KUKA KRL program: MyProgram_052().src

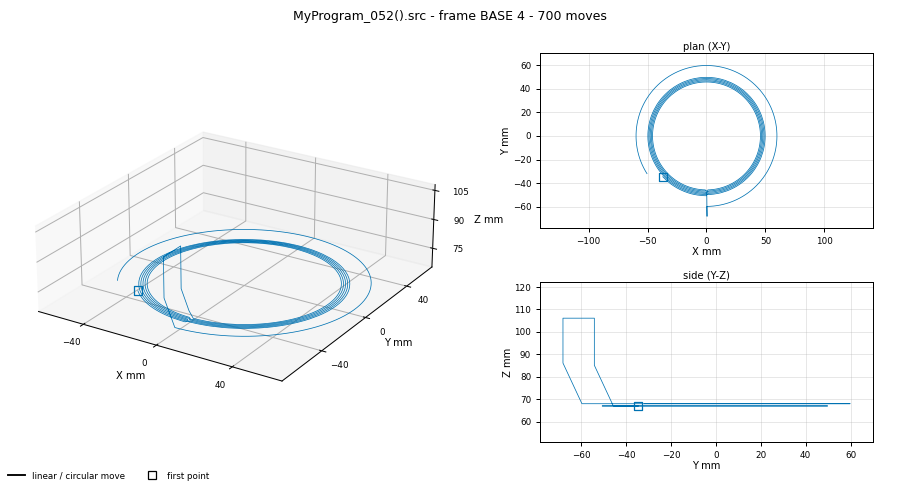
[picture p0: tool path of MyProgram_052().src in frame BASE 4, 700 of 700 moves have a stored position in this frame; points joined in program order, loops and branches not executed]
&ACCESS RVP
&REL 1
&PARAM TEMPLATE = C:\KRC\Roboter\Template\vorgabe
&PARAM EDITMASK = *
DEF MyProgram_052()
; ---- Setting reference (Base) ----
$BASE = BASE_DATA[4]

; --------------------------
; ---- Setting tool (TCP) ----
$TOOL = TOOL_DATA[3]
; --------------------------

$VEL.CP = VEL_APROX_PRINT
Startdeposition()
$VEL.CP = VEL_PRINT
LIN {X -37.0795,Y -34.6003,Z 67,A -142.3469,B 24.875,C -2.5805,E1 24.8845,E2 225.9733} C_DIS
LIN {X -35.1143,Y -36.5928,Z 67,A -139.506,B 24.8761,C -2.569,E1 24.8901,E2 223.1477} C_DIS
LIN {X -33.8275,Y -37.7853,Z 67,A -136.4507,B 24.8748,C -2.5821,E1 24.8966,E2 220.0491} C_DIS
LIN {X -30.4559,Y -40.5521,Z 67,A -131.9027,B 24.8763,C -2.5673,E1 24.9065,E2 215.5196} C_DIS
LIN {X -28.4082,Y -42.012,Z 67,A -128.4137,B 24.8757,C -2.5733,E1 24.9146,E2 212.0046} C_DIS
LIN {X -25.1167,Y -44.0592,Z 67,A -124.6294,B 24.8772,C -2.5574,E1 24.9237,E2 208.2469} C_DIS
LIN {X -22.6582,Y -45.3725,Z 67,A -121.2779,B 24.8772,C -2.5569,E1 24.9321,E2 204.8875} C_DIS
LIN {X -18.9408,Y -47.0459,Z 67,A -117.2171,B 24.8786,C -2.543,E1 24.9424,E2 200.8503} C_DIS
LIN {X -15.4527,Y -48.304,Z 67,A -112.4749,B 24.878,C -2.5491,E1 24.955,E2 196.0848} C_DIS
LIN {X -12.4723,Y -49.1576,Z 67,A -109.5038,B 24.8791,C -2.5379,E1 24.963,E2 193.1358} C_DIS
LIN {X -10.0949,Y -49.7005,Z 67,A -106.7826,B 24.8793,C -2.5361,E1 24.9704,E2 190.4157} C_DIS
LIN {X -7.4445,Y -50.1668,Z 67,A -103.2112,B 24.8785,C -2.5445,E1 24.9803,E2 186.8209} C_DIS
LIN {X -3.8911,Y -50.566,Z 67,A -100.05,B 24.88,C -2.5287,E1 24.989,E2 183.6956} C_DIS
LIN {X -2.1608,Y -50.6692,Z 67,A -97.7826,B 24.8794,C -2.5343,E1 24.9954,E2 181.4142} C_DIS
LIN {X -0.0557,Y -50.7153,Z 67,A -95.0288,B 24.8787,C -2.5416,E1 25.0031,E2 178.6432} C_DIS
LIN {X -0.0557,Y -50.7153,Z 67,A -95.0288,B 24.8787,C -2.5416,E1 25.0031,E2 178.6432} C_DIS
Enddeposition()
LIN {X 0.2505,Y -49.712,Z 67,A -95.9238,B 24.8792,C -2.5369,E1 25.0006,E2 179.5492} C_DIS
Startdeposition()
$VEL.CP = VEL_PRINT
LIN {X -2.7584,Y -49.6512,Z 67,A -99.9248,B 24.8801,C -2.5271,E1 24.9893,E2 183.5742} C_DIS
LIN {X -5.4391,Y -49.4301,Z 67,A -103.33,B 24.8806,C -2.5222,E1 24.9798,E2 186.9929} C_DIS
LIN {X -8.5864,Y -48.9804,Z 67,A -106.9223,B 24.8804,C -2.5244,E1 24.9699,E2 190.5832} C_DIS
LIN {X -12.0306,Y -48.2498,Z 67,A -110.567,B 24.8795,C -2.5331,E1 24.96,E2 194.212} C_DIS
LIN {X -15.2046,Y -47.3461,Z 67,A -115.2738,B 24.8807,C -2.5212,E1 24.9474,E2 198.9551} C_DIS
LIN {X -18.426,Y -46.1887,Z 67,A -119.1015,B 24.8802,C -2.5266,E1 24.9374,E2 202.778} C_DIS
LIN {X -22.1318,Y -44.5313,Z 67,A -122.9001,B 24.8783,C -2.5457,E1 24.9279,E2 206.5407} C_DIS
LIN {X -24.1155,Y -43.4892,Z 67,A -125.7875,B 24.8785,C -2.5443,E1 24.9208,E2 209.4396} C_DIS
LIN {X -27.878,Y -41.1784,Z 67,A -130.7372,B 24.8775,C -2.554,E1 24.9091,E2 214.382} C_DIS
LIN {X -29.9202,Y -39.7194,Z 67,A -133.864,B 24.8775,C -2.5552,E1 24.902,E2 217.5167} C_DIS
LIN {X -32.5332,Y -37.6097,Z 67,A -137.9216,B 24.877,C -2.5596,E1 24.8933,E2 221.5795} C_DIS
LIN {X -34.8779,Y -35.4455,Z 67,A -141.2483,B 24.8758,C -2.5721,E1 24.8866,E2 224.89} C_DIS
LIN {X -36.3763,Y -33.9066,Z 67,A -143.7227,B 24.8753,C -2.5774,E1 24.8819,E2 227.3625} C_DIS
LIN {X -37.7342,Y -32.3879,Z 67,A -145.936,B 24.8746,C -2.5845,E1 24.8778,E2 229.5687} C_DIS
LIN {X -38.7362,Y -31.183,Z 67,A -147.9222,B 24.8744,C -2.586,E1 24.8743,E2 231.5605} C_DIS
LIN {X -40.0423,Y -29.4865,Z 67,A -150.6165,B 24.8742,C -2.5886,E1 24.8697,E2 234.2615} C_DIS
LIN {X -42.0176,Y -26.5964,Z 67,A -154.4152,B 24.8729,C -2.6021,E1 24.8639,E2 238.0472} C_DIS
LIN {X -43.0644,Y -24.866,Z 67,A -157.367,B 24.8731,C -2.5994,E1 24.8597,E2 241.0208} C_DIS
LIN {X -44.6109,Y -21.9712,Z 67,A -160.8306,B 24.8717,C -2.614,E1 24.8553,E2 244.4679} C_DIS
LIN {X -45.6108,Y -19.8118,Z 67,A -163.4943,B 24.8708,C -2.6227,E1 24.8523,E2 247.1254} C_DIS
LIN {X -46.7007,Y -17.085,Z 67,A -166.8132,B 24.8698,C -2.6333,E1 24.849,E2 250.4376} C_DIS
LIN {X -47.5107,Y -14.6828,Z 67,A -170.2157,B 24.8696,C -2.6352,E1 24.8461,E2 253.855} C_DIS
LIN {X -48.4975,Y -10.9946,Z 67,A -173.9722,B 24.8674,C -2.6572,E1 24.8435,E2 257.5809} C_DIS
LIN {X -49.0589,Y -8.1285,Z 67,A -177.9765,B 24.8673,C -2.6587,E1 24.8415,E2 261.6052} C_DIS
LIN {X -49.4497,Y -5.2517,Z 67,A 179.0895,B 24.8657,C -2.6747,E1 24.8405,E2 264.5187} C_DIS
LIN {X -49.6264,Y -3.1776,Z 67,A 176.7448,B 24.8648,C -2.6829,E1 24.84,E2 266.8579} C_DIS
LIN {X -49.7186,Y -0.9552,Z 67,A 174.1077,B 24.8641,C -2.6899,E1 24.8398,E2 269.4941} C_DIS
LIN {X -49.6949,Y 1.8152,Z 67,A 170.5176,B 24.8636,C -2.6946,E1 24.84,E2 273.0947} C_DIS
LIN {X -49.522,Y 4.5195,Z 67,A 168.0202,B 24.8618,C -2.7128,E1 24.8405,E2 275.5633} C_DIS
LIN {X -49.2022,Y 7.208,Z 67,A 164.8184,B 24.8609,C -2.7215,E1 24.8416,E2 278.7635} C_DIS
LIN {X -48.9547,Y 8.7343,Z 67,A 162.6439,B 24.8609,C -2.7218,E1 24.8427,E2 280.9503} C_DIS
LIN {X -48.3657,Y 11.5613,Z 67,A 159.4302,B 24.8596,C -2.7336,E1 24.8446,E2 284.1545} C_DIS
LIN {X -47.5221,Y 14.646,Z 67,A 155.3988,B 24.859,C -2.7403,E1 24.8477,E2 288.1934} C_DIS
LIN {X -46.7485,Y 16.9539,Z 67,A 152.6347,B 24.858,C -2.7493,E1 24.8503,E2 290.9515} C_DIS
LIN {X -45.6266,Y 19.7752,Z 67,A 149.3564,B 24.8566,C -2.7627,E1 24.8538,E2 294.2159} C_DIS
LIN {X -44.6749,Y 21.8416,Z 67,A 146.0399,B 24.8568,C -2.7609,E1 24.8578,E2 297.5548} C_DIS
LIN {X -42.2626,Y 26.2058,Z 67,A 141.1281,B 24.8539,C -2.7886,E1 24.8646,E2 302.4259} C_DIS
LIN {X -40.6911,Y 28.5857,Z 67,A 136.9092,B 24.8544,C -2.7846,E1 24.8713,E2 306.6754} C_DIS
LIN {X -38.1447,Y 31.9031,Z 67,A 132.7078,B 24.8521,C -2.8056,E1 24.8785,E2 310.8463} C_DIS
LIN {X -36.5879,Y 33.6776,Z 67,A 130.0979,B 24.8513,C -2.8139,E1 24.8834,E2 313.448} C_DIS
LIN {X -35.0889,Y 35.2371,Z 67,A 127.5196,B 24.8508,C -2.8186,E1 24.8884,E2 316.0261} C_DIS
LIN {X -32.5963,Y 37.5546,Z 67,A 123.9843,B 24.8492,C -2.833,E1 24.8957,E2 319.5411} C_DIS
LIN {X -30.6979,Y 39.1218,Z 67,A 120.4276,B 24.8497,C -2.8286,E1 24.9035,E2 323.1218} C_DIS
LIN {X -28.804,Y 40.5362,Z 67,A 118.2528,B 24.8482,C -2.8421,E1 24.9083,E2 325.272} C_DIS
LIN {X -27.41,Y 41.4915,Z 67,A 115.4118,B 24.8493,C -2.8327,E1 24.915,E2 328.1448} C_DIS
LIN {X -23.7122,Y 43.7101,Z 67,A 110.8548,B 24.8477,C -2.8474,E1 24.926,E2 332.6803} C_DIS
LIN {X -20.8368,Y 45.1517,Z 67,A 107.4073,B 24.8466,C -2.857,E1 24.9346,E2 336.1138} C_DIS
LIN {X -18.9605,Y 45.9717,Z 67,A 104.6634,B 24.8469,C -2.8545,E1 24.9417,E2 338.87} C_DIS
LIN {X -15.5886,Y 47.2218,Z 67,A 100.8064,B 24.8459,C -2.864,E1 24.9518,E2 342.712} C_DIS
LIN {X -12.4514,Y 48.1437,Z 67,A 96.9923,B 24.8456,C -2.8672,E1 24.962,E2 346.5245} C_DIS
LIN {X -10.0971,Y 48.6919,Z 67,A 94.2114,B 24.8453,C -2.8696,E1 24.9696,E2 349.303} C_DIS
LIN {X -7.651,Y 49.1354,Z 67,A 91.5672,B 24.8447,C -2.8752,E1 24.9769,E2 351.9365} C_DIS
LIN {X -5.9044,Y 49.3761,Z 67,A 89.1599,B 24.8452,C -2.8703,E1 24.9836,E2 354.357} C_DIS
LIN {X -2.8923,Y 49.6437,Z 67,A 85.7598,B 24.8449,C -2.8732,E1 24.993,E2 357.7518} C_DIS
LIN {X -0.6646,Y 49.7234,Z 67,A 82.8665,B 24.8454,C -2.8686,E1 25.0011,E2 360.6563} C_DIS
LIN {X 2.8209,Y 49.6477,Z 67,A 78.8494,B 24.8454,C -2.8688,E1 25.0123,E2 364.6716} C_DIS
LIN {X 6.9409,Y 49.241,Z 67,A 75.0745,B 24.8436,C -2.8849,E1 25.0227,E2 368.4058} C_DIS
LIN {X 8.9379,Y 48.9175,Z 67,A 72.2375,B 24.8446,C -2.8755,E1 25.0306,E2 371.2623} C_DIS
LIN {X 12.2001,Y 48.2076,Z 67,A 67.5135,B 24.8465,C -2.8584,E1 25.0435,E2 376.0201} C_DIS
LIN {X 15.4724,Y 47.2597,Z 67,A 63.7622,B 24.8465,C -2.8584,E1 25.0535,E2 379.7645} C_DIS
LIN {X 19.2501,Y 45.8507,Z 67,A 60.0313,B 24.8452,C -2.8701,E1 25.0631,E2 383.4594} C_DIS
LIN {X 20.5782,Y 45.2704,Z 67,A 58.1872,B 24.8458,C -2.8651,E1 25.0678,E2 385.3108} C_DIS
LIN {X 22.4752,Y 44.3592,Z 67,A 54.4297,B 24.8486,C -2.8384,E1 25.0773,E2 389.1215} C_DIS
LIN {X 25.4752,Y 42.7072,Z 67,A 52.1521,B 24.846,C -2.8629,E1 25.0826,E2 391.3341} C_DIS
LIN {X 28.0765,Y 41.0441,Z 67,A 48.3054,B 24.8472,C -2.8521,E1 25.0917,E2 395.1939} C_DIS
LIN {X 29.9486,Y 39.6981,Z 67,A 45.4003,B 24.8482,C -2.843,E1 25.0982,E2 398.1102} C_DIS
LIN {X 32.0395,Y 38.0315,Z 67,A 41.483,B 24.8504,C -2.8218,E1 25.1067,E2 402.0627} C_DIS
LIN {X 34.3865,Y 35.9228,Z 67,A 37.8471,B 24.8512,C -2.8144,E1 25.1141,E2 405.701} C_DIS
LIN {X 37.3665,Y 32.8115,Z 67,A 33.7329,B 24.8507,C -2.8195,E1 25.1218,E2 409.7849} C_DIS
LIN {X 39.222,Y 30.5701,Z 67,A 30.767,B 24.8507,C -2.8192,E1 25.1269,E2 412.738} C_DIS
LIN {X 40.1847,Y 29.2925,Z 67,A 28.2929,B 24.8525,C -2.8026,E1 25.1311,E2 415.2393} C_DIS
LIN {X 42.0752,Y 26.5059,Z 67,A 24.9676,B 24.8524,C -2.8035,E1 25.1361,E2 418.5458} C_DIS
LIN {X 43.2785,Y 24.4929,Z 67,A 21.1417,B 24.8554,C -2.7747,E1 25.1415,E2 422.4201} C_DIS
LIN {X 44.8673,Y 21.4426,Z 67,A 17.9731,B 24.8549,C -2.7793,E1 25.1454,E2 425.5609} C_DIS
LIN {X 46.0689,Y 18.7215,Z 67,A 14.8326,B 24.8553,C -2.7753,E1 25.1488,E2 428.6938} C_DIS
LIN {X 46.7802,Y 16.8668,Z 67,A 12.2733,B 24.8566,C -2.7633,E1 25.1513,E2 431.267} C_DIS
LIN {X 47.7862,Y 13.7604,Z 67,A 9.0045,B 24.8567,C -2.762,E1 25.1539,E2 434.5203} C_DIS
LIN {X 48.2557,Y 12.0119,Z 67,A 6.634,B 24.8579,C -2.7501,E1 25.1556,E2 436.9052} C_DIS
LIN {X 48.8256,Y 9.4293,Z 67,A 3.4803,B 24.8591,C -2.7387,E1 25.1574,E2 440.0675} C_DIS
LIN {X 49.299,Y 6.5169,Z 67,A 0.1433,B 24.8601,C -2.7295,E1 25.1587,E2 443.4067} C_DIS
LIN {X 49.599,Y 3.5824,Z 67,A -3.0614,B 24.8608,C -2.7228,E1 25.1595,E2 446.6083} C_DIS
LIN {X 49.7259,Y 0.5187,Z 67,A -6.1684,B 24.861,C -2.7203,E1 25.1598,E2 449.7027} C_DIS
LIN {X 49.6721,Y -2.3404,Z 67,A -10.1157,B 24.8634,C -2.6968,E1 25.1594,E2 453.6821} C_DIS
LIN {X 49.4176,Y -5.5441,Z 67,A -13.6854,B 24.8643,C -2.6878,E1 25.1585,E2 457.2519} C_DIS
LIN {X 49.0237,Y -8.3395,Z 67,A -16.716,B 24.8649,C -2.682,E1 25.1572,E2 460.2784} C_DIS
LIN {X 48.5542,Y -10.7407,Z 67,A -19.5373,B 24.8658,C -2.6731,E1 25.1556,E2 463.1042} C_DIS
LIN {X 47.9955,Y -13.0107,Z 67,A -22.9399,B 24.8681,C -2.6507,E1 25.1531,E2 466.5404} C_DIS
LIN {X 46.3058,Y -18.128,Z 67,A -28.0338,B 24.8677,C -2.654,E1 25.1485,E2 471.5977} C_DIS
LIN {X 45.2339,Y -20.6589,Z 67,A -32.1672,B 24.8706,C -2.6254,E1 25.1438,E2 475.7762} C_DIS
LIN {X 43.2933,Y -24.4656,Z 67,A -36.6993,B 24.8712,C -2.619,E1 25.1378,E2 480.2998} C_DIS
LIN {X 41.4212,Y -27.5166,Z 67,A -40.1738,B 24.8711,C -2.6203,E1 25.1327,E2 483.7534} C_DIS
LIN {X 40.6509,Y -28.6409,Z 67,A -42.2645,B 24.8725,C -2.6059,E1 25.1293,E2 485.8682} C_DIS
LIN {X 38.573,Y -31.3844,Z 67,A -45.7048,B 24.8725,C -2.6057,E1 25.1234,E2 489.2925} C_DIS
LIN {X 36.6935,Y -33.5625,Z 67,A -49.7313,B 24.8747,C -2.5836,E1 25.1159,E2 493.3535} C_DIS
LIN {X 34.5074,Y -35.8063,Z 67,A -53.3041,B 24.8754,C -2.5757,E1 25.1088,E2 496.9298} C_DIS
LIN {X 31.3977,Y -38.5622,Z 67,A -57.3951,B 24.8752,C -2.5784,E1 25.1002,E2 500.9984} C_DIS
LIN {X 29.3776,Y -40.1224,Z 67,A -60.7741,B 24.8766,C -2.564,E1 25.0926,E2 504.3994} C_DIS
LIN {X 27.4879,Y -41.4401,Z 67,A -62.9553,B 24.8762,C -2.5677,E1 25.0876,E2 506.5643} C_DIS
LIN {X 25.4166,Y -42.7418,Z 67,A -66.3813,B 24.8778,C -2.5512,E1 25.0794,E2 510.0189} C_DIS
LIN {X 23.1942,Y -43.9872,Z 67,A -68.7496,B 24.8773,C -2.5567,E1 25.0736,E2 512.3672} C_DIS
LIN {X 19.9272,Y -45.5605,Z 67,A -73.7738,B 24.8794,C -2.5348,E1 25.0608,E2 517.4306} C_DIS
LIN {X 17.454,Y -46.5643,Z 67,A -77.1022,B 24.8802,C -2.5261,E1 25.0521,E2 520.7725} C_DIS
LIN {X 12.1079,Y -48.2312,Z 67,A -82.4712,B 24.879,C -2.5385,E1 25.0378,E2 526.1029} C_DIS
LIN {X 10.0818,Y -48.6949,Z 67,A -85.0863,B 24.8796,C -2.5324,E1 25.0306,E2 528.729} C_DIS
LIN {X 7.4223,Y -49.171,Z 67,A -87.7994,B 24.8792,C -2.5372,E1 25.0232,E2 531.428} C_DIS
LIN {X 6.033,Y -49.3603,Z 67,A -89.9034,B 24.8801,C -2.5276,E1 25.0173,E2 533.5531} C_DIS
LIN {X 3.1793,Y -49.6263,Z 67,A -93.4479,B 24.8806,C -2.5219,E1 25.0074,E2 537.1095} C_DIS
LIN {X 0.2505,Y -49.712,Z 67,A -95.9232,B 24.8792,C -2.5367,E1 25.0006,E2 539.5492} C_DIS
Enddeposition()
LIN {X 0.2505,Y -49.712,Z 67,A -95.9232,B 24.8792,C -2.5367,E1 25.0006,E2 539.5492} C_DIS
Startdeposition()
$VEL.CP = VEL_PRINT
LIN {X 1.4593,Y -48.7184,Z 67,A -93.5201,B 24.8759,C -2.5709,E1 25.0075,E2 537.0653} C_DIS
LIN {X 3.9754,Y -48.5779,Z 67,A -90.7627,B 24.8761,C -2.5686,E1 25.0152,E2 534.3145} C_DIS
LIN {X 6.1747,Y -48.3476,Z 67,A -88.2241,B 24.8761,C -2.5691,E1 25.0222,E2 531.7766} C_DIS
LIN {X 9.1506,Y -47.8736,Z 67,A -83.9458,B 24.8746,C -2.5849,E1 25.034,E2 527.4652} C_DIS
LIN {X 14.099,Y -46.6564,Z 67,A -77.8877,B 24.8738,C -2.5924,E1 25.0504,E2 521.3992} C_DIS
LIN {X 17.6898,Y -45.417,Z 67,A -73.6014,B 24.8736,C -2.5949,E1 25.0616,E2 517.116} C_DIS
LIN {X 21.6587,Y -43.6636,Z 67,A -69.008,B 24.8737,C -2.5933,E1 25.0732,E2 512.5382} C_DIS
LIN {X 24.0511,Y -42.3932,Z 67,A -65.7906,B 24.8731,C -2.5993,E1 25.0811,E2 509.3158} C_DIS
LIN {X 26.2006,Y -41.0994,Z 67,A -62.4617,B 24.8719,C -2.612,E1 25.089,E2 505.9674} C_DIS
LIN {X 29.7642,Y -38.5967,Z 67,A -57.7772,B 24.8717,C -2.6141,E1 25.0995,E2 501.2945} C_DIS
LIN {X 32.7938,Y -36.0568,Z 67,A -52.8175,B 24.8701,C -2.6305,E1 25.11,E2 496.3155} C_DIS
LIN {X 35.5576,Y -33.3335,Z 67,A -47.8569,B 24.8682,C -2.6494,E1 25.1197,E2 491.3315} C_DIS
LIN {X 38.127,Y -30.364,Z 67,A -43.4377,B 24.8674,C -2.6573,E1 25.1275,E2 486.9139} C_DIS
LIN {X 40.6831,Y -26.842,Z 67,A -38.9979,B 24.8674,C -2.6578,E1 25.1346,E2 482.4949} C_DIS
LIN {X 42.0184,Y -24.6997,Z 67,A -36.0839,B 24.8666,C -2.665,E1 25.1388,E2 479.5785} C_DIS
LIN {X 43.3733,Y -22.2345,Z 67,A -33.2124,B 24.8666,C -2.6659,E1 25.1426,E2 476.72} C_DIS
LIN {X 44.4214,Y -20.0587,Z 67,A -29.4695,B 24.8639,C -2.6923,E1 25.1471,E2 472.9349} C_DIS
LIN {X 45.6985,Y -16.9491,Z 67,A -25.6028,B 24.8628,C -2.7025,E1 25.151,E2 469.0656} C_DIS
LIN {X 46.9143,Y -13.216,Z 67,A -21.4414,B 24.8623,C -2.7075,E1 25.1544,E2 464.916} C_DIS
LIN {X 47.7125,Y -9.9576,Z 67,A -17.156,B 24.8604,C -2.7267,E1 25.157,E2 460.6102} C_DIS
LIN {X 48.2077,Y -7.1897,Z 67,A -14.3099,B 24.8603,C -2.7278,E1 25.1583,E2 457.7781} C_DIS
LIN {X 48.4802,Y -5.0283,Z 67,A -11.7765,B 24.8595,C -2.7353,E1 25.1591,E2 455.2419} C_DIS
LIN {X 48.6854,Y -2.3119,Z 67,A -8.1781,B 24.8576,C -2.7534,E1 25.1597,E2 451.6221} C_DIS
LIN {X 48.7412,Y 0.2134,Z 67,A -5.2697,B 24.8568,C -2.7615,E1 25.1597,E2 448.712} C_DIS
LIN {X 48.6356,Y 3.1938,Z 67,A -1.9945,B 24.8561,C -2.7678,E1 25.1593,E2 445.4412} C_DIS
LIN {X 48.4596,Y 5.2249,Z 67,A 0.2962,B 24.8555,C -2.7732,E1 25.1586,E2 443.1514} C_DIS
LIN {X 47.9146,Y 8.9375,Z 67,A 4.6496,B 24.8543,C -2.7855,E1 25.1567,E2 438.7943} C_DIS
LIN {X 47.2883,Y 11.8111,Z 67,A 8.1227,B 24.8531,C -2.7963,E1 25.1545,E2 435.3159} C_DIS
LIN {X 46.5524,Y 14.4391,Z 67,A 11.526,B 24.8517,C -2.8097,E1 25.1518,E2 431.9005} C_DIS
LIN {X 45.5852,Y 17.251,Z 67,A 14.5058,B 24.8517,C -2.8095,E1 25.149,E2 428.9376} C_DIS
LIN {X 44.771,Y 19.267,Z 67,A 17.3201,B 24.8504,C -2.8218,E1 25.146,E2 426.1097} C_DIS
LIN {X 43.9622,Y 21.0462,Z 67,A 19.3244,B 24.8504,C -2.8224,E1 25.1436,E2 424.1148} C_DIS
LIN {X 42.5457,Y 23.7797,Z 67,A 23.1875,B 24.8488,C -2.8369,E1 25.1386,E2 420.2378} C_DIS
LIN {X 41.3344,Y 25.8279,Z 67,A 25.7483,B 24.8485,C -2.8395,E1 25.1349,E2 417.6839} C_DIS
LIN {X 40.3728,Y 27.3066,Z 67,A 28.4737,B 24.8466,C -2.8573,E1 25.1306,E2 414.9297} C_DIS
LIN {X 38.5139,Y 29.8716,Z 67,A 32.2504,B 24.8455,C -2.8672,E1 25.1242,E2 411.1476} C_DIS
LIN {X 36.3063,Y 32.5187,Z 67,A 35.8708,B 24.8455,C -2.868,E1 25.1176,E2 407.5417} C_DIS
LIN {X 33.6815,Y 35.2308,Z 67,A 40.9102,B 24.8432,C -2.8887,E1 25.1076,E2 402.4747} C_DIS
LIN {X 30.8052,Y 37.7713,Z 67,A 44.786,B 24.8436,C -2.8852,E1 25.0994,E2 398.6222} C_DIS
LIN {X 28.1121,Y 39.8168,Z 67,A 48.2961,B 24.8438,C -2.8834,E1 25.0915,E2 395.1288} C_DIS
LIN {X 25.7687,Y 41.3714,Z 67,A 51.6887,B 24.8431,C -2.8901,E1 25.0836,E2 391.7315} C_DIS
LIN {X 24.4467,Y 42.1658,Z 67,A 53.8882,B 24.842,C -2.8997,E1 25.0782,E2 389.5159} C_DIS
LIN {X 21.4963,Y 43.7441,Z 67,A 57.6781,B 24.8417,C -2.9021,E1 25.0689,E2 385.7308} C_DIS
LIN {X 19.4392,Y 44.696,Z 67,A 60.07,B 24.842,C -2.9002,E1 25.0628,E2 383.3494} C_DIS
LIN {X 17.4937,Y 45.4922,Z 67,A 63.0781,B 24.8406,C -2.9121,E1 25.0549,E2 380.3197} C_DIS
LIN {X 14.4878,Y 46.5373,Z 67,A 66.272,B 24.8414,C -2.9055,E1 25.0465,E2 377.1476} C_DIS
LIN {X 12.305,Y 47.161,Z 67,A 69.2063,B 24.8407,C -2.9118,E1 25.0386,E2 374.203} C_DIS
LIN {X 9.7775,Y 47.7495,Z 67,A 72.2311,B 24.8406,C -2.9129,E1 25.0303,E2 371.1797} C_DIS
LIN {X 7.2536,Y 48.1976,Z 67,A 75.2551,B 24.8404,C -2.914,E1 25.022,E2 368.1561} C_DIS
LIN {X 4.5447,Y 48.5279,Z 67,A 78.6127,B 24.8401,C -2.917,E1 25.0127,E2 364.7937} C_DIS
LIN {X 1.7948,Y 48.7077,Z 67,A 81.8002,B 24.8402,C -2.916,E1 25.0038,E2 361.6096} C_DIS
LIN {X -0.4565,Y 48.7383,Z 67,A 84.1756,B 24.8408,C -2.911,E1 24.9972,E2 359.2462} C_DIS
LIN {X -2.6649,Y 48.6673,Z 67,A 86.9936,B 24.8405,C -2.9138,E1 24.9893,E2 356.4211} C_DIS
LIN {X -4.7797,Y 48.5057,Z 67,A 89.5773,B 24.8405,C -2.914,E1 24.9821,E2 353.8354} C_DIS
LIN {X -6.6855,Y 48.2795,Z 67,A 91.8359,B 24.8405,C -2.9127,E1 24.9759,E2 351.5782} C_DIS
LIN {X -9.959,Y 47.7122,Z 67,A 96.0485,B 24.8404,C -2.9145,E1 24.9643,E2 347.3566} C_DIS
LIN {X -14.1936,Y 46.6285,Z 67,A 100.7637,B 24.8417,C -2.9026,E1 24.9517,E2 342.6626} C_DIS
LIN {X -16.3104,Y 45.9305,Z 67,A 103.2846,B 24.8422,C -2.898,E1 24.945,E2 340.1479} C_DIS
LIN {X -18.2361,Y 45.2004,Z 67,A 106.0304,B 24.842,C -2.8997,E1 24.9379,E2 337.392} C_DIS
LIN {X -21.0515,Y 43.9595,Z 67,A 109.3865,B 24.843,C -2.8904,E1 24.9294,E2 334.0498} C_DIS
LIN {X -23.0132,Y 42.9659,Z 67,A 112.6518,B 24.8424,C -2.8964,E1 24.9213,E2 330.7611} C_DIS
LIN {X -27.1404,Y 40.4849,Z 67,A 117.4332,B 24.8449,C -2.873,E1 24.91,E2 326.0207} C_DIS
LIN {X -29.6729,Y 38.667,Z 67,A 122.0754,B 24.8442,C -2.8799,E1 24.8995,E2 321.3454} C_DIS
LIN {X -32.0865,Y 36.6888,Z 67,A 125.4244,B 24.8455,C -2.8672,E1 24.8925,E2 318.0138} C_DIS
LIN {X -34.5849,Y 34.3437,Z 67,A 128.9159,B 24.8474,C -2.8501,E1 24.8855,E2 314.5485} C_DIS
LIN {X -35.6779,Y 33.206,Z 67,A 131.5205,B 24.8467,C -2.8563,E1 24.8805,E2 311.9176} C_DIS
LIN {X -38.542,Y 29.8352,Z 67,A 135.6777,B 24.8497,C -2.8284,E1 24.8732,E2 307.8081} C_DIS
LIN {X -39.8556,Y 28.0576,Z 67,A 139.4151,B 24.8488,C -2.8374,E1 24.867,E2 304.031} C_DIS
LIN {X -41.2946,Y 25.8916,Z 67,A 141.8914,B 24.8505,C -2.8208,E1 24.8633,E2 301.5817} C_DIS
LIN {X -42.2826,Y 24.2435,Z 67,A 144.4806,B 24.8507,C -2.8191,E1 24.8597,E2 298.9832} C_DIS
LIN {X -43.9141,Y 21.1462,Z 67,A 148.3951,B 24.8523,C -2.8044,E1 24.8548,E2 295.0829} C_DIS
LIN {X -44.9155,Y 18.9264,Z 67,A 151.2125,B 24.8532,C -2.7953,E1 24.8516,E2 292.2717} C_DIS
LIN {X -45.8241,Y 16.6065,Z 67,A 153.896,B 24.8545,C -2.7831,E1 24.849,E2 289.6021} C_DIS
LIN {X -46.5695,Y 14.3838,Z 67,A 157.4063,B 24.8543,C -2.785,E1 24.846,E2 286.0673} C_DIS
LIN {X -47.4055,Y 11.3304,Z 67,A 160.3577,B 24.8566,C -2.763,E1 24.844,E2 283.1512} C_DIS
LIN {X -47.7895,Y 9.5786,Z 67,A 162.6746,B 24.857,C -2.7593,E1 24.8426,E2 280.8297} C_DIS
LIN {X -48.2667,Y 6.7781,Z 67,A 166.8386,B 24.857,C -2.7601,E1 24.8408,E2 276.639} C_DIS
LIN {X -48.6347,Y 3.2063,Z 67,A 170.7388,B 24.8587,C -2.7424,E1 24.84,E2 272.7577} C_DIS
LIN {X -48.7424,Y 0.0227,Z 67,A 174.5122,B 24.8599,C -2.731,E1 24.8398,E2 268.9889} C_DIS
LIN {X -48.6213,Y -3.4029,Z 67,A 178.1219,B 24.8618,C -2.7127,E1 24.8403,E2 265.4012} C_DIS
LIN {X -48.4408,Y -5.3948,Z 67,A -179.255,B 24.8622,C -2.7091,E1 24.841,E2 262.7709} C_DIS
LIN {X -48.0762,Y -8.0162,Z 67,A -176.3395,B 24.8634,C -2.6969,E1 24.8423,E2 259.8673} C_DIS
LIN {X -47.5785,Y -10.5799,Z 67,A -172.8888,B 24.8638,C -2.6928,E1 24.8442,E2 256.406} C_DIS
LIN {X -46.7055,Y -13.9359,Z 67,A -169.0415,B 24.8654,C -2.6775,E1 24.8471,E2 252.5729} C_DIS
LIN {X -45.9885,Y -16.1451,Z 67,A -166.1966,B 24.866,C -2.6711,E1 24.8496,E2 249.727} C_DIS
LIN {X -44.665,Y -19.5103,Z 67,A -161.662,B 24.8668,C -2.6631,E1 24.8545,E2 245.1864} C_DIS
LIN {X -43.2186,Y -22.5344,Z 67,A -157.8085,B 24.868,C -2.6512,E1 24.8593,E2 241.3407} C_DIS
LIN {X -41.6168,Y -25.3705,Z 67,A -153.8406,B 24.8688,C -2.6432,E1 24.8649,E2 237.3712} C_DIS
LIN {X -40.1943,Y -27.5702,Z 67,A -151.3138,B 24.8704,C -2.6276,E1 24.8688,E2 234.8692} C_DIS
LIN {X -38.8864,Y -29.3846,Z 67,A -148.356,B 24.8705,C -2.626,E1 24.8737,E2 231.9008} C_DIS
LIN {X -37.3702,Y -31.2907,Z 67,A -145.5748,B 24.8713,C -2.6183,E1 24.8786,E2 229.1253} C_DIS
LIN {X -35.6731,Y -33.2129,Z 67,A -142.3396,B 24.8716,C -2.615,E1 24.8847,E2 225.8837} C_DIS
LIN {X -33.8634,Y -35.0555,Z 67,A -139.6153,B 24.8727,C -2.6041,E1 24.89,E2 223.1737} C_DIS
LIN {X -32.2252,Y -36.5675,Z 67,A -136.7648,B 24.8728,C -2.6025,E1 24.896,E2 220.3158} C_DIS
LIN {X -30.3831,Y -38.112,Z 67,A -133.7171,B 24.873,C -2.6007,E1 24.9026,E2 217.2608} C_DIS
LIN {X -27.5312,Y -40.2207,Z 67,A -129.8182,B 24.8741,C -2.5897,E1 24.9114,E2 213.3746} C_DIS
LIN {X -24.555,Y -42.1039,Z 67,A -125.5983,B 24.8746,C -2.5849,E1 24.9215,E2 209.153} C_DIS
LIN {X -23.107,Y -42.915,Z 67,A -123.4273,B 24.8745,C -2.5858,E1 24.9268,E2 206.9737} C_DIS
LIN {X -20.4141,Y -44.2595,Z 67,A -119.7902,B 24.8747,C -2.5833,E1 24.936,E2 203.3333} C_DIS
LIN {X -17.4239,Y -45.5198,Z 67,A -116.5653,B 24.876,C -2.5702,E1 24.9443,E2 200.1325} C_DIS
LIN {X -15.5468,Y -46.1942,Z 67,A -113.8882,B 24.8757,C -2.5736,E1 24.9514,E2 197.442} C_DIS
LIN {X -12.8352,Y -47.02,Z 67,A -110.5462,B 24.8758,C -2.5716,E1 24.9604,E2 194.0994} C_DIS
LIN {X -9.4545,Y -47.8151,Z 67,A -105.9303,B 24.8752,C -2.5787,E1 24.973,E2 189.4611} C_DIS
LIN {X -5.6403,Y -48.4128,Z 67,A -101.9402,B 24.8761,C -2.5685,E1 24.984,E2 185.492} C_DIS
LIN {X -2.9306,Y -48.6526,Z 67,A -99.0645,B 24.8767,C -2.563,E1 24.992,E2 182.6282} C_DIS
LIN {X -1.0392,Y -48.7294,Z 67,A -96.7997,B 24.8766,C -2.564,E1 24.9983,E2 180.3608} C_DIS
LIN {X 0.2379,Y -48.7342,Z 67,A -95.3358,B 24.8766,C -2.5638,E1 25.0024,E2 178.8975} C_DIS
Enddeposition()
LIN {X 0.2379,Y -48.7342,Z 67,A -95.3358,B 24.8766,C -2.5638,E1 25.0024,E2 178.8975} C_DIS
Startdeposition()
$VEL.CP = VEL_PRINT
LIN {X -0.8805,Y -47.7446,Z 67,A -97.8451,B 24.8769,C -2.561,E1 24.9954,E2 181.4134} C_DIS
LIN {X -3.3224,Y -47.6371,Z 67,A -100.7978,B 24.8769,C -2.5605,E1 24.9871,E2 184.3681} C_DIS
LIN {X -5.768,Y -47.4036,Z 67,A -103.7394,B 24.8769,C -2.5609,E1 24.9789,E2 187.3105} C_DIS
LIN {X -8.6463,Y -46.9639,Z 67,A -107.7465,B 24.8776,C -2.5539,E1 24.9679,E2 191.3382} C_DIS
LIN {X -12.3361,Y -46.132,Z 67,A -111.6373,B 24.8764,C -2.5664,E1 24.9574,E2 195.2047} C_DIS
LIN {X -15.4067,Y -45.1994,Z 67,A -115.1387,B 24.8756,C -2.5745,E1 24.9481,E2 198.6927} C_DIS
LIN {X -17.9717,Y -44.2419,Z 67,A -118.9673,B 24.8761,C -2.5692,E1 24.938,E2 202.542} C_DIS
LIN {X -21.0789,Y -42.8489,Z 67,A -122.9705,B 24.8755,C -2.575,E1 24.9279,E2 206.5414} C_DIS
LIN {X -22.4857,Y -42.1282,Z 67,A -124.9714,B 24.8755,C -2.5759,E1 24.923,E2 208.5459} C_DIS
LIN {X -25.2515,Y -40.5301,Z 67,A -128.6188,B 24.8746,C -2.584,E1 24.9142,E2 212.1849} C_DIS
LIN {X -26.8598,Y -39.4827,Z 67,A -131.226,B 24.8747,C -2.5832,E1 24.9081,E2 214.8028} C_DIS
LIN {X -29.3649,Y -37.6577,Z 67,A -134.5088,B 24.8735,C -2.5958,E1 24.9008,E2 218.0671} C_DIS
LIN {X -31.275,Y -36.0862,Z 67,A -137.9785,B 24.8737,C -2.5941,E1 24.8934,E2 221.5541} C_DIS
LIN {X -33.3426,Y -34.1846,Z 67,A -141.3462,B 24.873,C -2.6009,E1 24.8866,E2 224.9196} C_DIS
LIN {X -34.97,Y -32.5192,Z 67,A -143.7846,B 24.8719,C -2.6118,E1 24.8819,E2 227.3426} C_DIS
LIN {X -36.4873,Y -30.8059,Z 67,A -146.7887,B 24.8717,C -2.6143,E1 24.8764,E2 230.3541} C_DIS
LIN {X -37.9974,Y -28.9223,Z 67,A -149.7426,B 24.8711,C -2.6203,E1 24.8713,E2 233.3077} C_DIS
LIN {X -39.0395,Y -27.5013,Z 67,A -151.7547,B 24.8704,C -2.6268,E1 24.8681,E2 235.3141} C_DIS
LIN {X -40.9376,Y -24.5855,Z 67,A -156.3462,B 24.8699,C -2.6319,E1 24.8612,E2 239.9169} C_DIS
LIN {X -42.3573,Y -22.0507,Z 67,A -159.1053,B 24.8681,C -2.6508,E1 24.8576,E2 242.6452} C_DIS
LIN {X -43.1053,Y -20.5493,Z 67,A -161.6755,B 24.8682,C -2.6489,E1 24.8544,E2 245.234} C_DIS
LIN {X -44.2989,Y -17.8315,Z 67,A -164.6864,B 24.8665,C -2.6662,E1 24.8511,E2 248.2202} C_DIS
LIN {X -45.2199,Y -15.3458,Z 67,A -168.2612,B 24.8661,C -2.6701,E1 24.8477,E2 251.8058} C_DIS
LIN {X -45.9403,Y -13.0314,Z 67,A -171.8862,B 24.8661,C -2.6695,E1 24.8449,E2 255.4534} C_DIS
LIN {X -46.6754,Y -10.0866,Z 67,A -175.843,B 24.8655,C -2.6764,E1 24.8425,E2 259.4167} C_DIS
LIN {X -47.5276,Y -4.6383,Z 67,A 177.5165,B 24.8634,C -2.6966,E1 24.8402,E2 266.0488} C_DIS
LIN {X -47.7544,Y 0.123,Z 67,A 172.5012,B 24.8607,C -2.7234,E1 24.8398,E2 271.03} C_DIS
LIN {X -47.6492,Y 3.1444,Z 67,A 168.9744,B 24.8594,C -2.7362,E1 24.8403,E2 274.5476} C_DIS
LIN {X -47.4199,Y 5.6286,Z 67,A 165.7581,B 24.8587,C -2.7427,E1 24.8412,E2 277.7674} C_DIS
LIN {X -46.9854,Y 8.5266,Z 67,A 162.3283,B 24.8575,C -2.7548,E1 24.8428,E2 281.1887} C_DIS
LIN {X -46.4595,Y 11.0418,Z 67,A 159.1989,B 24.8565,C -2.7638,E1 24.8447,E2 284.315} C_DIS
LIN {X -45.4398,Y 14.6815,Z 67,A 154.9667,B 24.8547,C -2.7816,E1 24.848,E2 288.5289} C_DIS
LIN {X -44.837,Y 16.4309,Z 67,A 152.2795,B 24.8546,C -2.7823,E1 24.8506,E2 291.2297} C_DIS
LIN {X -43.5109,Y 19.6756,Z 67,A 148.6833,B 24.8524,C -2.8027,E1 24.8544,E2 294.7971} C_DIS
LIN {X -42.7705,Y 21.237,Z 67,A 145.603,B 24.8532,C -2.7957,E1 24.8583,E2 297.9108} C_DIS
LIN {X -40.4326,Y 25.4076,Z 67,A 141.0462,B 24.8498,C -2.8273,E1 24.8646,E2 302.4158} C_DIS
LIN {X -39.6242,Y 26.6508,Z 67,A 137.8079,B 24.8514,C -2.8129,E1 24.8697,E2 305.7045} C_DIS
LIN {X -37.8385,Y 29.1303,Z 67,A 134.4133,B 24.85,C -2.8261,E1 24.8754,E2 309.0839} C_DIS
LIN {X -34.9965,Y 32.4907,Z 67,A 129.6965,B 24.8477,C -2.8468,E1 24.884,E2 313.7726} C_DIS
LIN {X -32.7743,Y 34.73,Z 67,A 125.6223,B 24.8472,C -2.8517,E1 24.8921,E2 317.852} C_DIS
LIN {X -30.7953,Y 36.4969,Z 67,A 121.4253,B 24.8479,C -2.845,E1 24.9012,E2 322.0814} C_DIS
LIN {X -28.2041,Y 38.5338,Z 67,A 119.3844,B 24.8442,C -2.8794,E1 24.9055,E2 324.0474} C_DIS
LIN {X -25.5987,Y 40.3122,Z 67,A 114.9364,B 24.8444,C -2.8773,E1 24.9159,E2 328.5151} C_DIS
LIN {X -23.557,Y 41.5385,Z 67,A 111.8608,B 24.8442,C -2.8792,E1 24.9233,E2 331.5954} C_DIS
LIN {X -21.2684,Y 42.7549,Z 67,A 108.9001,B 24.8435,C -2.8864,E1 24.9306,E2 334.5471} C_DIS
LIN {X -19.0839,Y 43.7736,Z 67,A 106.2711,B 24.8426,C -2.8945,E1 24.9373,E2 337.1633} C_DIS
LIN {X -17.4659,Y 44.444,Z 67,A 104.1059,B 24.8424,C -2.8964,E1 24.9429,E2 339.3287} C_DIS
LIN {X -15.3136,Y 45.2308,Z 67,A 101.032,B 24.8425,C -2.895,E1 24.951,E2 342.4119} C_DIS
LIN {X -12.2362,Y 46.1582,Z 67,A 97.2173,B 24.842,C -2.8997,E1 24.9612,E2 346.2217} C_DIS
LIN {X -10.3338,Y 46.6215,Z 67,A 95.1716,B 24.8413,C -2.9063,E1 24.9667,E2 348.2542} C_DIS
LIN {X -8.1342,Y 47.0554,Z 67,A 91.9166,B 24.842,C -2.8998,E1 24.9757,E2 351.5282} C_DIS
LIN {X -5.7055,Y 47.4109,Z 67,A 89.5753,B 24.8408,C -2.9109,E1 24.9821,E2 353.8449} C_DIS
LIN {X -2.9652,Y 47.6602,Z 67,A 85.6281,B 24.8417,C -2.9023,E1 24.9932,E2 357.8142} C_DIS
LIN {X 0.1509,Y 47.7525,Z 67,A 82.0269,B 24.8414,C -2.9054,E1 25.0032,E2 361.4082} C_DIS
LIN {X 2.4181,Y 47.692,Z 67,A 79.6585,B 24.8408,C -2.9111,E1 25.0098,E2 363.7623} C_DIS
LIN {X 4.2599,Y 47.5625,Z 67,A 77.4326,B 24.8408,C -2.9109,E1 25.016,E2 365.9876} C_DIS
LIN {X 7.2119,Y 47.205,Z 67,A 73.0104,B 24.8424,C -2.8962,E1 25.0283,E2 370.4408} C_DIS
LIN {X 12.3617,Y 46.1251,Z 67,A 67.3075,B 24.8416,C -2.903,E1 25.0438,E2 376.1197} C_DIS
LIN {X 14.8947,Y 45.3708,Z 67,A 64.2308,B 24.8417,C -2.9022,E1 25.0519,E2 379.1928} C_DIS
LIN {X 18.0981,Y 44.1904,Z 67,A 60.1231,B 24.8422,C -2.8982,E1 25.0627,E2 383.3012} C_DIS
LIN {X 19.9801,Y 43.3723,Z 67,A 57.7407,B 24.8423,C -2.8968,E1 25.0687,E2 385.6809} C_DIS
LIN {X 22.8837,Y 41.9123,Z 67,A 54.0533,B 24.8425,C -2.8956,E1 25.0779,E2 389.361} C_DIS
LIN {X 24.318,Y 41.0969,Z 67,A 51.9384,B 24.843,C -2.8904,E1 25.083,E2 391.4817} C_DIS
LIN {X 26.0678,Y 40.0099,Z 67,A 49.3468,B 24.8437,C -2.8846,E1 25.0891,E2 394.0789} C_DIS
LIN {X 28.3239,Y 38.4456,Z 67,A 45.5512,B 24.8452,C -2.8702,E1 25.0978,E2 397.8952} C_DIS
LIN {X 30.6342,Y 36.6319,Z 67,A 42.5657,B 24.8449,C -2.8734,E1 25.1042,E2 400.862} C_DIS
LIN {X 32.9764,Y 34.5388,Z 67,A 38.4766,B 24.8463,C -2.8601,E1 25.1126,E2 404.9658} C_DIS
LIN {X 35.6597,Y 31.7604,Z 67,A 34.2996,B 24.8465,C -2.8585,E1 25.1206,E2 409.1285} C_DIS
LIN {X 37.0006,Y 30.1874,Z 67,A 31.6747,B 24.8474,C -2.8502,E1 25.1253,E2 411.7611} C_DIS
LIN {X 38.2289,Y 28.6161,Z 67,A 29.3186,B 24.8479,C -2.8451,E1 25.1292,E2 414.1179} C_DIS
LIN {X 39.349,Y 27.0562,Z 67,A 27.0348,B 24.8485,C -2.8398,E1 25.1329,E2 416.403} C_DIS
LIN {X 40.6603,Y 25.0429,Z 67,A 24.2286,B 24.8491,C -2.8339,E1 25.1371,E2 419.2091} C_DIS
LIN {X 41.813,Y 23.0664,Z 67,A 21.2216,B 24.8504,C -2.8218,E1 25.1412,E2 422.2292} C_DIS
LIN {X 43.5227,Y 19.6493,Z 67,A 17.2484,B 24.8505,C -2.8208,E1 25.1461,E2 426.1834} C_DIS
LIN {X 44.1118,Y 18.2906,Z 67,A 15.1502,B 24.8517,C -2.8097,E1 25.1484,E2 428.2965} C_DIS
LIN {X 44.9782,Y 16.0419,Z 67,A 11.5404,B 24.854,C -2.7878,E1 25.1518,E2 431.9379} C_DIS
LIN {X 46.1763,Y 12.1721,Z 67,A 7.791,B 24.8533,C -2.7946,E1 25.1548,E2 435.6498} C_DIS
LIN {X 46.794,Y 9.521,Z 67,A 4.1386,B 24.8551,C -2.7773,E1 25.157,E2 439.3219} C_DIS
LIN {X 47.3267,Y 6.3687,Z 67,A 0.3276,B 24.8563,C -2.7659,E1 25.1586,E2 443.1373} C_DIS
LIN {X 47.591,Y 3.9285,Z 67,A -2.5629,B 24.8571,C -2.7578,E1 25.1594,E2 446.0298} C_DIS
LIN {X 47.73,Y 1.4746,Z 67,A -5.4353,B 24.858,C -2.7501,E1 25.1597,E2 448.9035} C_DIS
LIN {X 47.749,Y -0.6452,Z 67,A -7.8052,B 24.8584,C -2.7454,E1 25.1597,E2 451.2703} C_DIS
LIN {X 47.6821,Y -2.5965,Z 67,A -10.294,B 24.8595,C -2.7352,E1 25.1594,E2 453.7685} C_DIS
LIN {X 47.5418,Y -4.4845,Z 67,A -12.3497,B 24.8598,C -2.7323,E1 25.1589,E2 455.8189} C_DIS
LIN {X 47.2954,Y -6.5943,Z 67,A -15.195,B 24.8612,C -2.7185,E1 25.1579,E2 458.68} C_DIS
LIN {X 46.9361,Y -8.7935,Z 67,A -17.6525,B 24.8616,C -2.7143,E1 25.1567,E2 461.133} C_DIS
LIN {X 46.5221,Y -10.7712,Z 67,A -20.2147,B 24.8627,C -2.7041,E1 25.1552,E2 463.7046} C_DIS
LIN {X 45.869,Y -13.2829,Z 67,A -23.9383,B 24.8648,C -2.6827,E1 25.1524,E2 467.4573} C_DIS
LIN {X 44.4034,Y -17.5691,Z 67,A -28.5756,B 24.865,C -2.6816,E1 25.148,E2 472.0714} C_DIS
LIN {X 42.937,Y -20.8996,Z 67,A -32.8257,B 24.866,C -2.6709,E1 25.1431,E2 476.3236} C_DIS
LIN {X 41.5741,Y -23.4933,Z 67,A -36.7771,B 24.8679,C -2.6525,E1 25.1378,E2 480.2979} C_DIS
LIN {X 40.3467,Y -25.5449,Z 67,A -39.1194,B 24.8677,C -2.6545,E1 25.1344,E2 482.6236} C_DIS
LIN {X 39.2475,Y -27.2023,Z 67,A -41.7993,B 24.8689,C -2.6424,E1 25.1302,E2 485.3188} C_DIS
LIN {X 38.0099,Y -28.9074,Z 67,A -44.0866,B 24.8691,C -2.6402,E1 25.1264,E2 487.6003} C_DIS
LIN {X 36.6643,Y -30.5951,Z 67,A -46.8265,B 24.8701,C -2.6307,E1 25.1215,E2 490.35} C_DIS
LIN {X 34.5175,Y -32.9971,Z 67,A -50.6698,B 24.871,C -2.6216,E1 25.1143,E2 494.198} C_DIS
LIN {X 32.6584,Y -34.8391,Z 67,A -54.0669,B 24.8722,C -2.6094,E1 25.1074,E2 497.6096} C_DIS
LIN {X 30.8927,Y -36.414,Z 67,A -56.6212,B 24.8722,C -2.6084,E1 25.102,E2 500.1565} C_DIS
LIN {X 28.5289,Y -38.2934,Z 67,A -60.1071,B 24.8728,C -2.6033,E1 25.0943,E2 503.6417} C_DIS
LIN {X 26.6259,Y -39.6411,Z 67,A -63.0452,B 24.8736,C -2.5952,E1 25.0875,E2 506.589} C_DIS
LIN {X 24.9244,Y -40.7323,Z 67,A -65.1525,B 24.8734,C -2.5964,E1 25.0826,E2 508.6866} C_DIS
LIN {X 22.8784,Y -41.9156,Z 67,A -68.1666,B 24.8742,C -2.5882,E1 25.0752,E2 511.7111} C_DIS
LIN {X 20.6788,Y -43.0431,Z 67,A -72.0177,B 24.8762,C -2.5679,E1 25.0655,E2 515.6003} C_DIS
LIN {X 16.4757,Y -44.8207,Z 67,A -76.5978,B 24.8754,C -2.576,E1 25.0537,E2 520.1508} C_DIS
LIN {X 14.4501,Y -45.5142,Z 67,A -79.1669,B 24.8757,C -2.5729,E1 25.0469,E2 522.7224} C_DIS
LIN {X 12.0104,Y -46.2179,Z 67,A -82.3103,B 24.8762,C -2.568,E1 25.0384,E2 525.8722} C_DIS
LIN {X 8.4385,Y -47.0012,Z 67,A -86.3364,B 24.876,C -2.5704,E1 25.0274,E2 529.8876} C_DIS
LIN {X 6.9973,Y -47.2381,Z 67,A -88.565,B 24.8769,C -2.5611,E1 25.0212,E2 532.1362} C_DIS
LIN {X 4.0279,Y -47.5831,Z 67,A -92.0175,B 24.8769,C -2.5614,E1 25.0116,E2 535.5857} C_DIS
LIN {X 1.7579,Y -47.7211,Z 67,A -94.5788,B 24.8767,C -2.5631,E1 25.0045,E2 538.1421} C_DIS
LIN {X 0.2387,Y -47.7456,Z 67,A -96.133,B 24.8763,C -2.5672,E1 25.0002,E2 539.6864} C_DIS
Enddeposition()
LIN {X 0.2387,Y -47.7456,Z 67,A -96.133,B 24.8763,C -2.5672,E1 25.0002,E2 539.6864} C_DIS
Startdeposition()
$VEL.CP = VEL_PRINT
LIN {X 1.8327,Y -46.7294,Z 67,A -93.2127,B 24.873,C -2.6008,E1 25.0085,E2 536.6869} C_DIS
LIN {X 4.9175,Y -46.506,Z 67,A -89.2039,B 24.8725,C -2.6064,E1 25.0197,E2 532.667} C_DIS
LIN {X 7.5812,Y -46.1469,Z 67,A -85.4961,B 24.8715,C -2.6158,E1 25.03,E2 528.9404} C_DIS
LIN {X 10.9752,Y -45.4593,Z 67,A -81.7825,B 24.8721,C -2.6105,E1 25.0401,E2 525.2443} C_DIS
LIN {X 13.3642,Y -44.8151,Z 67,A -78.809,B 24.8718,C -2.6128,E1 25.0481,E2 522.2704} C_DIS
LIN {X 15.4576,Y -44.1367,Z 67,A -75.2612,B 24.87,C -2.6312,E1 25.0575,E2 518.6861} C_DIS
LIN {X 18.6683,Y -42.8775,Z 67,A -71.8728,B 24.8709,C -2.6222,E1 25.0662,E2 515.3268} C_DIS
LIN {X 21.0957,Y -41.7373,Z 67,A -68.5502,B 24.8703,C -2.6281,E1 25.0745,E2 511.9992} C_DIS
LIN {X 22.7199,Y -40.8755,Z 67,A -65.9123,B 24.8692,C -2.6389,E1 25.081,E2 509.3432} C_DIS
LIN {X 25.3597,Y -39.2923,Z 67,A -62.1198,B 24.8685,C -2.6464,E1 25.09,E2 505.5452} C_DIS
LIN {X 29.0551,Y -36.6442,Z 67,A -57.1259,B 24.8685,C -2.6472,E1 25.1011,E2 500.5673} C_DIS
LIN {X 31.0194,Y -34.9977,Z 67,A -54.0349,B 24.8678,C -2.6533,E1 25.1077,E2 497.474} C_DIS
LIN {X 33.0016,Y -33.1349,Z 67,A -50.3718,B 24.8664,C -2.6673,E1 25.115,E2 493.7931} C_DIS
LIN {X 35.107,Y -30.8953,Z 67,A -46.9282,B 24.8661,C -2.6705,E1 25.1215,E2 490.357} C_DIS
LIN {X 36.7575,Y -28.9117,Z 67,A -43.7225,B 24.8652,C -2.6795,E1 25.1271,E2 487.1448} C_DIS
LIN {X 38.0321,Y -27.213,Z 67,A -41.0872,B 24.8644,C -2.6871,E1 25.1315,E2 484.5043} C_DIS
LIN {X 39.4083,Y -25.1791,Z 67,A -37.5911,B 24.8626,C -2.7048,E1 25.1368,E2 480.984} C_DIS
LIN {X 41.6744,Y -21.2188,Z 67,A -32.5966,B 24.8621,C -2.7093,E1 25.1435,E2 476.0048} C_DIS
LIN {X 42.9572,Y -18.4855,Z 67,A -28.9059,B 24.861,C -2.7201,E1 25.1477,E2 472.3087} C_DIS
LIN {X 44.2766,Y -15.0528,Z 67,A -24.5185,B 24.8599,C -2.7314,E1 25.152,E2 467.9191} C_DIS
LIN {X 44.9495,Y -12.9058,Z 67,A -21.841,B 24.8592,C -2.7384,E1 25.1541,E2 465.2403} C_DIS
LIN {X 45.5125,Y -10.7545,Z 67,A -19.1571,B 24.8584,C -2.746,E1 25.1559,E2 462.5539} C_DIS
LIN {X 46.0045,Y -8.4016,Z 67,A -16.1669,B 24.8573,C -2.7561,E1 25.1575,E2 459.5573} C_DIS
LIN {X 46.2782,Y -6.7337,Z 67,A -13.3103,B 24.855,C -2.7779,E1 25.1587,E2 456.6659} C_DIS
LIN {X 46.6312,Y -3.5429,Z 67,A -10.2432,B 24.8555,C -2.7734,E1 25.1595,E2 453.6276} C_DIS
LIN {X 46.7523,Y -1.131,Z 67,A -7.1667,B 24.8543,C -2.785,E1 25.1598,E2 450.5419} C_DIS
LIN {X 46.7418,Y 1.4825,Z 67,A -4.1755,B 24.8537,C -2.791,E1 25.1596,E2 447.5544} C_DIS
LIN {X 46.6064,Y 3.8533,Z 67,A -1.1483,B 24.8525,C -2.8024,E1 25.159,E2 444.5183} C_DIS
LIN {X 46.3406,Y 6.2945,Z 67,A 1.8904,B 24.8514,C -2.8122,E1 25.158,E2 441.4742} C_DIS
LIN {X 45.9103,Y 8.9013,Z 67,A 5.8323,B 24.8489,C -2.8358,E1 25.156,E2 437.4996} C_DIS
LIN {X 44.7784,Y 13.4878,Z 67,A 11.1672,B 24.848,C -2.8442,E1 25.1521,E2 432.1754} C_DIS
LIN {X 43.8107,Y 16.3602,Z 67,A 14.4843,B 24.8477,C -2.8474,E1 25.149,E2 428.8695} C_DIS
LIN {X 42.9082,Y 18.598,Z 67,A 17.3477,B 24.847,C -2.854,E1 25.1459,E2 426.0063} C_DIS
LIN {X 42.1365,Y 20.2857,Z 67,A 19.8206,B 24.8459,C -2.864,E1 25.1429,E2 423.5229} C_DIS
LIN {X 40.8744,Y 22.7218,Z 67,A 22.8566,B 24.8456,C -2.8668,E1 25.1389,E2 420.4962} C_DIS
LIN {X 39.6691,Y 24.766,Z 67,A 25.9707,B 24.8444,C -2.8782,E1 25.1344,E2 417.371} C_DIS
LIN {X 38.2133,Y 26.9591,Z 67,A 29.0972,B 24.8437,C -2.8844,E1 25.1295,E2 414.2453} C_DIS
LIN {X 36.8129,Y 28.8413,Z 67,A 32.1597,B 24.8426,C -2.8947,E1 25.1242,E2 411.173} C_DIS
LIN {X 35.0131,Y 31.0022,Z 67,A 35.3861,B 24.8422,C -2.8984,E1 25.1184,E2 407.9524} C_DIS
LIN {X 33.0809,Y 33.0563,Z 67,A 38.9782,B 24.8411,C -2.9082,E1 25.1114,E2 404.3524} C_DIS
LIN {X 31.0758,Y 34.9472,Z 67,A 42.154,B 24.8407,C -2.9112,E1 25.1049,E2 401.1823} C_DIS
LIN {X 29.1943,Y 36.5342,Z 67,A 45.3561,B 24.8398,C -2.9201,E1 25.0979,E2 397.9713} C_DIS
LIN {X 26.6824,Y 38.4063,Z 67,A 48.4762,B 24.8405,C -2.9139,E1 25.0909,E2 394.877} C_DIS
LIN {X 24.8836,Y 39.5956,Z 67,A 51.8102,B 24.8387,C -2.9301,E1 25.0831,E2 391.5155} C_DIS
LIN {X 22.5234,Y 40.984,Z 67,A 55.1348,B 24.8382,C -2.9342,E1 25.075,E2 388.1911} C_DIS
LIN {X 19.9269,Y 42.3078,Z 67,A 58.4377,B 24.8382,C -2.9339,E1 25.0667,E2 384.8977} C_DIS
LIN {X 18.1019,Y 43.1198,Z 67,A 60.6493,B 24.8384,C -2.9325,E1 25.0611,E2 382.6948} C_DIS
LIN {X 16.2494,Y 43.8521,Z 67,A 63.504,B 24.8374,C -2.9418,E1 25.0536,E2 379.8242} C_DIS
LIN {X 13.805,Y 44.6812,Z 67,A 66.6238,B 24.8372,C -2.9435,E1 25.0453,E2 376.706} C_DIS
LIN {X 11.309,Y 45.3778,Z 67,A 69.3239,B 24.8378,C -2.9376,E1 25.0381,E2 374.0242} C_DIS
LIN {X 9.2518,Y 45.8412,Z 67,A 72.4241,B 24.8368,C -2.9473,E1 25.0296,E2 370.905} C_DIS
LIN {X 7.0053,Y 46.2378,Z 67,A 74.7931,B 24.8374,C -2.9413,E1 25.0231,E2 368.5527} C_DIS
LIN {X 4.2365,Y 46.573,Z 67,A 78.2461,B 24.8373,C -2.9424,E1 25.0135,E2 365.0995} C_DIS
LIN {X 2.8041,Y 46.6816,Z 67,A 80.7448,B 24.836,C -2.9542,E1 25.0065,E2 362.5738} C_DIS
LIN {X -0.9401,Y 46.7559,Z 67,A 84.8767,B 24.8369,C -2.9462,E1 24.995,E2 358.4613} C_DIS
LIN {X -4.176,Y 46.5786,Z 67,A 88.9543,B 24.8369,C -2.9462,E1 24.9836,E2 354.3821} C_DIS
LIN {X -6.8066,Y 46.2678,Z 67,A 92.0822,B 24.8373,C -2.9424,E1 24.975,E2 351.2609} C_DIS
LIN {X -9.4288,Y 45.8049,Z 67,A 95.4719,B 24.8373,C -2.9418,E1 24.9657,E2 347.8689} C_DIS
LIN {X -12.123,Y 45.1665,Z 67,A 98.9796,B 24.8375,C -2.9403,E1 24.9562,E2 344.3597} C_DIS
LIN {X -14.7811,Y 44.3682,Z 67,A 102.2837,B 24.8381,C -2.935,E1 24.9474,E2 341.0624} C_DIS
LIN {X -17.2195,Y 43.4798,Z 67,A 105.4606,B 24.8386,C -2.9309,E1 24.9391,E2 337.8888} C_DIS
LIN {X -19.1962,Y 42.6438,Z 67,A 108.6381,B 24.8381,C -2.935,E1 24.931,E2 334.6937} C_DIS
LIN {X -21.9218,Y 41.3091,Z 67,A 112.4652,B 24.8386,C -2.9306,E1 24.9215,E2 330.8667} C_DIS
LIN {X -25.6477,Y 39.1049,Z 67,A 117.1725,B 24.8406,C -2.9124,E1 24.9104,E2 326.188} C_DIS
LIN {X -28.2964,Y 37.234,Z 67,A 120.7103,B 24.8421,C -2.8984,E1 24.9025,E2 322.6713} C_DIS
LIN {X -30.1587,Y 35.742,Z 67,A 124.0333,B 24.8422,C -2.8977,E1 24.8952,E2 319.3375} C_DIS
LIN {X -32.4432,Y 33.6813,Z 67,A 127.8627,B 24.8431,C -2.8899,E1 24.8874,E2 315.5111} C_DIS
LIN {X -34.2616,Y 31.8309,Z 67,A 131.0695,B 24.8439,C -2.8826,E1 24.8812,E2 312.3078} C_DIS
LIN {X -35.5999,Y 30.3255,Z 67,A 134.2236,B 24.8435,C -2.8857,E1 24.8755,E2 309.132} C_DIS
LIN {X -37.4208,Y 28.0477,Z 67,A 137.2137,B 24.8454,C -2.8686,E1 24.8704,E2 306.1687} C_DIS
LIN {X -38.9017,Y 25.9559,Z 67,A 140.2811,B 24.8464,C -2.8591,E1 24.8656,E2 303.1087} C_DIS
LIN {X -40.529,Y 23.3322,Z 67,A 144.4725,B 24.847,C -2.8539,E1 24.8596,E2 298.908} C_DIS
LIN {X -42.0016,Y 20.5647,Z 67,A 147.8901,B 24.8488,C -2.8373,E1 24.8553,E2 295.512} C_DIS
LIN {X -43.0007,Y 18.3845,Z 67,A 150.7007,B 24.8499,C -2.827,E1 24.8521,E2 292.7106} C_DIS
LIN {X -43.8499,Y 16.2553,Z 67,A 153.8873,B 24.8502,C -2.8234,E1 24.8489,E2 289.5145} C_DIS
LIN {X -44.7939,Y 13.4355,Z 67,A 157.576,B 24.8514,C -2.8129,E1 24.8458,E2 285.8299} C_DIS
LIN {X -45.558,Y 10.5572,Z 67,A 161.1268,B 24.8527,C -2.8003,E1 24.8434,E2 282.2883} C_DIS
LIN {X -46.0007,Y 8.4228,Z 67,A 164.0592,B 24.8532,C -2.7954,E1 24.8419,E2 279.3505} C_DIS
LIN {X -46.4342,Y 5.556,Z 67,A 167.2651,B 24.8549,C -2.7798,E1 24.8407,E2 276.1627} C_DIS
LIN {X -46.6495,Y 3.2907,Z 67,A 170.0954,B 24.8557,C -2.7716,E1 24.84,E2 273.3351} C_DIS
LIN {X -46.7617,Y 0.6196,Z 67,A 173.4073,B 24.8567,C -2.7617,E1 24.8398,E2 270.0269} C_DIS
LIN {X -46.7123,Y -2.2364,Z 67,A 176.9362,B 24.8578,C -2.7511,E1 24.8401,E2 266.5019} C_DIS
LIN {X -46.518,Y -4.803,Z 67,A -179.7886,B 24.8587,C -2.7429,E1 24.8409,E2 263.2268} C_DIS
LIN {X -46.2565,Y -6.8838,Z 67,A -177.1084,B 24.8594,C -2.7364,E1 24.8419,E2 260.5461} C_DIS
LIN {X -45.7055,Y -9.8994,Z 67,A -173.5583,B 24.8608,C -2.7224,E1 24.8438,E2 257.0087} C_DIS
LIN {X -45.0834,Y -12.4311,Z 67,A -170.1387,B 24.8615,C -2.7158,E1 24.8463,E2 253.5849} C_DIS
LIN {X -44.3883,Y -14.7213,Z 67,A -167.1835,B 24.8623,C -2.7075,E1 24.8488,E2 250.6326} C_DIS
LIN {X -43.5953,Y -16.9256,Z 67,A -164.3424,B 24.8632,C -2.6989,E1 24.8516,E2 247.796} C_DIS
LIN {X -42.5577,Y -19.3874,Z 67,A -160.9972,B 24.864,C -2.6907,E1 24.8553,E2 244.452} C_DIS
LIN {X -41.4961,Y -21.5669,Z 67,A -158.5396,B 24.8655,C -2.6758,E1 24.8584,E2 242.0168} C_DIS
LIN {X -40.0907,Y -24.0788,Z 67,A -154.5688,B 24.8659,C -2.6726,E1 24.8639,E2 238.0331} C_DIS
LIN {X -38.7645,Y -26.1592,Z 67,A -151.5165,B 24.8666,C -2.6654,E1 24.8686,E2 234.9825} C_DIS
LIN {X -37.2568,Y -28.2661,Z 67,A -148.5897,B 24.8677,C -2.6544,E1 24.8734,E2 232.0679} C_DIS
LIN {X -36.1254,Y -29.6983,Z 67,A -146.0406,B 24.8677,C -2.6536,E1 24.8779,E2 229.5089} C_DIS
LIN {X -34.1562,Y -31.9431,Z 67,A -141.5678,B 24.8674,C -2.6571,E1 24.8864,E2 225.0079} C_DIS
LIN {X -31.5864,Y -34.4861,Z 67,A -136.9257,B 24.868,C -2.6514,E1 24.8959,E2 220.3605} C_DIS
LIN {X -28.3829,Y -37.1677,Z 67,A -132.8257,B 24.8704,C -2.6274,E1 24.9047,E2 216.3024} C_DIS
LIN {X -26.1884,Y -38.7448,Z 67,A -129.4804,B 24.8709,C -2.6226,E1 24.9124,E2 212.9572} C_DIS
LIN {X -23.8997,Y -40.1965,Z 67,A -126.189,B 24.8714,C -2.6173,E1 24.9202,E2 209.6681} C_DIS
LIN {X -21.9206,Y -41.3098,Z 67,A -123.5748,B 24.872,C -2.6112,E1 24.9266,E2 207.0611} C_DIS
LIN {X -20.5524,Y -42.0077,Z 67,A -121.4139,B 24.8718,C -2.6131,E1 24.932,E2 204.8899} C_DIS
LIN {X -18.1444,Y -43.1018,Z 67,A -118.2293,B 24.8722,C -2.6089,E1 24.9402,E2 201.7079} C_DIS
LIN {X -15.724,Y -44.0433,Z 67,A -115.0177,B 24.8724,C -2.6065,E1 24.9486,E2 198.4953} C_DIS
LIN {X -14.0729,Y -44.5982,Z 67,A -112.6206,B 24.8722,C -2.609,E1 24.955,E2 196.0879} C_DIS
LIN {X -11.1118,Y -45.426,Z 67,A -109.5491,B 24.8735,C -2.596,E1 24.9632,E2 193.0429} C_DIS
LIN {X -8.0558,Y -46.0667,Z 67,A -105.3558,B 24.8731,C -2.6002,E1 24.9747,E2 188.8347} C_DIS
LIN {X -5.9329,Y -46.3875,Z 67,A -102.8481,B 24.8733,C -2.5977,E1 24.9817,E2 186.331} C_DIS
LIN {X -3.9886,Y -46.5956,Z 67,A -100.1636,B 24.8729,C -2.6022,E1 24.9892,E2 183.6344} C_DIS
LIN {X -1.1721,Y -46.7513,Z 67,A -97.2401,B 24.8737,C -2.5939,E1 24.9973,E2 180.7302} C_DIS
LIN {X 0.2268,Y -46.7486,Z 67,A -95.4675,B 24.8735,C -2.5955,E1 25.0022,E2 178.9537} C_DIS
Enddeposition()
LIN {X 0.2268,Y -46.7486,Z 67,A -95.4675,B 24.8735,C -2.5955,E1 25.0022,E2 178.9537} C_DIS
Startdeposition()
$VEL.CP = VEL_PRINT
LIN {X -1.1279,Y -45.7647,Z 67,A -98.262,B 24.8736,C -2.5944,E1 24.9944,E2 181.7508} C_DIS
LIN {X -3.3084,Y -45.6586,Z 67,A -101.0163,B 24.8736,C -2.594,E1 24.9867,E2 184.5071} C_DIS
LIN {X -5.6016,Y -45.4346,Z 67,A -103.8197,B 24.8736,C -2.5955,E1 24.979,E2 187.3085} C_DIS
LIN {X -7.7383,Y -45.1194,Z 67,A -106.6368,B 24.8736,C -2.5946,E1 24.9712,E2 190.1305} C_DIS
LIN {X -9.984,Y -44.6764,Z 67,A -109.4753,B 24.8735,C -2.5962,E1 24.9634,E2 192.9685} C_DIS
LIN {X -12.1511,Y -44.1362,Z 67,A -112.2827,B 24.8733,C -2.5976,E1 24.9558,E2 195.7768} C_DIS
LIN {X -14.3662,Y -43.466,Z 67,A -115.1307,B 24.873,C -2.6004,E1 24.9483,E2 198.623} C_DIS
LIN {X -16.4765,Y -42.7107,Z 67,A -117.9646,B 24.8728,C -2.6025,E1 24.9408,E2 201.4579} C_DIS
LIN {X -18.492,Y -41.8771,Z 67,A -120.7229,B 24.8726,C -2.6049,E1 24.9337,E2 204.2168} C_DIS
LIN {X -20.5875,Y -40.888,Z 67,A -123.5877,B 24.8722,C -2.6088,E1 24.9266,E2 207.0798} C_DIS
LIN {X -22.5132,Y -39.8599,Z 67,A -126.408,B 24.872,C -2.6111,E1 24.9197,E2 209.9025} C_DIS
LIN {X -24.4697,Y -38.6898,Z 67,A -129.2112,B 24.8715,C -2.616,E1 24.913,E2 212.7029} C_DIS
LIN {X -26.3235,Y -37.4531,Z 67,A -132.037,B 24.8711,C -2.6199,E1 24.9065,E2 215.5288} C_DIS
LIN {X -28.166,Y -36.0882,Z 67,A -134.8924,B 24.8706,C -2.625,E1 24.9001,E2 218.3823} C_DIS
LIN {X -29.9748,Y -34.5998,Z 67,A -137.9811,B 24.8703,C -2.6284,E1 24.8935,E2 221.475} C_DIS
LIN {X -31.7708,Y -32.9579,Z 67,A -140.9085,B 24.8695,C -2.636,E1 24.8876,E2 224.3961} C_DIS
LIN {X -33.3293,Y -31.3809,Z 67,A -143.7051,B 24.869,C -2.6416,E1 24.8822,E2 227.1915} C_DIS
LIN {X -34.516,Y -30.0708,Z 67,A -146.0111,B 24.8686,C -2.6452,E1 24.8779,E2 229.4992} C_DIS
LIN {X -36.079,Y -28.1776,Z 67,A -148.9904,B 24.8678,C -2.6535,E1 24.8727,E2 232.4725} C_DIS
LIN {X -37.4296,Y -26.3572,Z 67,A -151.8448,B 24.8671,C -2.6602,E1 24.868,E2 235.325} C_DIS
LIN {X -38.6725,Y -24.4973,Z 67,A -154.6498,B 24.8664,C -2.6671,E1 24.8638,E2 238.1275} C_DIS
LIN {X -39.8225,Y -22.5796,Z 67,A -157.4643,B 24.8657,C -2.6742,E1 24.8598,E2 240.9397} C_DIS
LIN {X -40.8901,Y -20.5835,Z 67,A -160.3378,B 24.865,C -2.6813,E1 24.8561,E2 243.8115} C_DIS
LIN {X -41.8247,Y -18.6103,Z 67,A -163.0924,B 24.8643,C -2.6886,E1 24.8529,E2 246.5638} C_DIS
LIN {X -42.7125,Y -16.4718,Z 67,A -166.0041,B 24.8634,C -2.6966,E1 24.8499,E2 249.4725} C_DIS
LIN {X -43.4487,Y -14.4173,Z 67,A -168.7766,B 24.8627,C -2.704,E1 24.8474,E2 252.2431} C_DIS
LIN {X -44.1192,Y -12.2137,Z 67,A -171.6383,B 24.8618,C -2.7128,E1 24.8451,E2 255.1004} C_DIS
LIN {X -44.6665,Y -10.0291,Z 67,A -174.4857,B 24.861,C -2.7209,E1 24.8433,E2 257.9451} C_DIS
LIN {X -45.1077,Y -7.8084,Z 67,A -177.3193,B 24.8601,C -2.7295,E1 24.8418,E2 260.7748} C_DIS
LIN {X -45.4351,Y -5.5976,Z 67,A 179.8364,B 24.8592,C -2.7376,E1 24.8408,E2 263.6168} C_DIS
LIN {X -45.6542,Y -3.3726,Z 67,A 177.0344,B 24.8583,C -2.7462,E1 24.8401,E2 266.4149} C_DIS
LIN {X -45.7643,Y -1.1402,Z 67,A 174.2675,B 24.8574,C -2.7554,E1 24.8398,E2 269.1767} C_DIS
LIN {X -45.7654,Y 1.0917,Z 67,A 171.365,B 24.8566,C -2.7628,E1 24.8398,E2 272.0788} C_DIS
LIN {X -45.6585,Y 3.3097,Z 67,A 168.5612,B 24.8557,C -2.7713,E1 24.8404,E2 274.8792} C_DIS
LIN {X -45.4349,Y 5.5989,Z 67,A 165.6823,B 24.8548,C -2.7803,E1 24.8412,E2 277.7538} C_DIS
LIN {X -45.1167,Y 7.7544,Z 67,A 162.9032,B 24.854,C -2.7882,E1 24.8425,E2 280.5305} C_DIS
LIN {X -44.6785,Y 9.974,Z 67,A 160.0607,B 24.8531,C -2.7969,E1 24.8441,E2 283.3689} C_DIS
LIN {X -44.1364,Y 12.1504,Z 67,A 157.1889,B 24.8522,C -2.8048,E1 24.8461,E2 286.2387} C_DIS
LIN {X -43.4553,Y 14.3978,Z 67,A 154.3393,B 24.8512,C -2.8148,E1 24.8485,E2 289.0805} C_DIS
LIN {X -42.7035,Y 16.4948,Z 67,A 151.493,B 24.8503,C -2.8225,E1 24.8513,E2 291.9246} C_DIS
LIN {X -41.8728,Y 18.502,Z 67,A 148.73,B 24.8495,C -2.83,E1 24.8543,E2 294.6848} C_DIS
LIN {X -40.8936,Y 20.5764,Z 67,A 145.8803,B 24.8486,C -2.8386,E1 24.8578,E2 297.5294} C_DIS
LIN {X -39.8712,Y 22.4929,Z 67,A 143.1019,B 24.8479,C -2.8456,E1 24.8615,E2 300.3057} C_DIS
LIN {X -38.7516,Y 24.3708,Z 67,A 140.3335,B 24.8471,C -2.8528,E1 24.8656,E2 303.071} C_DIS
LIN {X -37.4664,Y 26.3043,Z 67,A 137.4221,B 24.8463,C -2.8606,E1 24.8701,E2 305.9782} C_DIS
LIN {X -36.076,Y 28.1814,Z 67,A 134.5062,B 24.8454,C -2.8684,E1 24.8751,E2 308.8895} C_DIS
LIN {X -34.6571,Y 29.9092,Z 67,A 131.6905,B 24.8447,C -2.8752,E1 24.8801,E2 311.7018} C_DIS
LIN {X -33.1545,Y 31.5668,Z 67,A 128.8814,B 24.8439,C -2.8819,E1 24.8854,E2 314.5072} C_DIS
LIN {X -31.5725,Y 33.149,Z 67,A 125.9318,B 24.8434,C -2.8865,E1 24.8913,E2 317.4581} C_DIS
LIN {X -29.7107,Y 34.8264,Z 67,A 122.8937,B 24.8425,C -2.8948,E1 24.8977,E2 320.4885} C_DIS
LIN {X -27.7823,Y 36.3839,Z 67,A 119.957,B 24.8416,C -2.9034,E1 24.9041,E2 323.4153} C_DIS
LIN {X -26.2654,Y 37.4935,Z 67,A 117.4492,B 24.8413,C -2.9061,E1 24.9098,E2 325.9256} C_DIS
LIN {X -24.4468,Y 38.7041,Z 67,A 114.7286,B 24.8407,C -2.9113,E1 24.9162,E2 328.6424} C_DIS
LIN {X -22.5476,Y 39.8406,Z 67,A 111.9269,B 24.8402,C -2.9158,E1 24.9229,E2 331.442} C_DIS
LIN {X -20.5887,Y 40.8875,Z 67,A 109.085,B 24.8398,C -2.9194,E1 24.93,E2 334.2829} C_DIS
LIN {X -18.5943,Y 41.8319,Z 67,A 106.3314,B 24.8394,C -2.9236,E1 24.9369,E2 337.0333} C_DIS
LIN {X -16.4677,Y 42.7141,Z 67,A 103.4419,B 24.839,C -2.9274,E1 24.9444,E2 339.9202} C_DIS
LIN {X -14.4143,Y 43.4498,Z 67,A 100.6811,B 24.8386,C -2.9303,E1 24.9517,E2 342.6794} C_DIS
LIN {X -12.155,Y 44.1351,Z 67,A 97.7948,B 24.8382,C -2.9344,E1 24.9594,E2 345.5606} C_DIS
LIN {X -9.9977,Y 44.6734,Z 67,A 94.9911,B 24.8379,C -2.9366,E1 24.967,E2 348.3627} C_DIS
LIN {X -7.8106,Y 45.1073,Z 67,A 92.1851,B 24.8377,C -2.9385,E1 24.9747,E2 351.1671} C_DIS
LIN {X -5.6016,Y 45.4346,Z 67,A 89.3585,B 24.8376,C -2.9398,E1 24.9826,E2 353.993} C_DIS
LIN {X -3.3788,Y 45.6537,Z 67,A 86.5587,B 24.8375,C -2.941,E1 24.9903,E2 356.7912} C_DIS
LIN {X -1.009,Y 45.7669,Z 67,A 83.6892,B 24.8372,C -2.9434,E1 24.9983,E2 359.6554} C_DIS
LIN {X 1.2068,Y 45.7623,Z 67,A 80.847,B 24.8372,C -2.9428,E1 25.0063,E2 362.4988} C_DIS
LIN {X 3.3095,Y 45.6585,Z 67,A 78.1309,B 24.8374,C -2.9416,E1 25.0138,E2 365.2167} C_DIS
LIN {X 5.6231,Y 45.4318,Z 67,A 75.2719,B 24.8374,C -2.9419,E1 25.0218,E2 368.0729} C_DIS
LIN {X 7.7739,Y 45.1134,Z 67,A 72.5272,B 24.8374,C -2.9407,E1 25.0293,E2 370.8178} C_DIS
LIN {X 9.982,Y 44.6768,Z 67,A 69.7081,B 24.8376,C -2.9394,E1 25.037,E2 373.6364} C_DIS
LIN {X 12.0386,Y 44.1666,Z 67,A 67.0061,B 24.8379,C -2.937,E1 25.0443,E2 376.3399} C_DIS
LIN {X 14.3595,Y 43.4682,Z 67,A 64.0751,B 24.8379,C -2.9363,E1 25.0521,E2 379.2671} C_DIS
LIN {X 16.4699,Y 42.7132,Z 67,A 61.2475,B 24.8383,C -2.9334,E1 25.0595,E2 382.0957} C_DIS
LIN {X 18.5008,Y 41.8733,Z 67,A 58.5222,B 24.8386,C -2.931,E1 25.0665,E2 384.8203} C_DIS
LIN {X 20.4214,Y 40.9705,Z 67,A 55.7256,B 24.8392,C -2.9255,E1 25.0736,E2 387.6226} C_DIS
LIN {X 22.5832,Y 39.8205,Z 67,A 52.7839,B 24.8394,C -2.9234,E1 25.0808,E2 390.5607} C_DIS
LIN {X 24.4651,Y 38.6927,Z 67,A 50.0753,B 24.8398,C -2.92,E1 25.0872,E2 393.2689} C_DIS
LIN {X 26.3066,Y 37.4648,Z 67,A 47.2529,B 24.8404,C -2.9146,E1 25.0937,E2 396.0943} C_DIS
LIN {X 28.3498,Y 35.9429,Z 67,A 44.1047,B 24.8409,C -2.9098,E1 25.1007,E2 399.2426} C_DIS
LIN {X 30.0884,Y 34.5006,Z 67,A 41.2819,B 24.8415,C -2.9045,E1 25.1067,E2 402.0669} C_DIS
LIN {X 31.9119,Y 32.8219,Z 67,A 38.0552,B 24.8424,C -2.8961,E1 25.1133,E2 405.3002} C_DIS
LIN {X 33.8201,Y 30.8517,Z 67,A 34.6965,B 24.8431,C -2.89,E1 25.1197,E2 408.6587} C_DIS
LIN {X 35.562,Y 28.8262,Z 67,A 31.4816,B 24.8436,C -2.8847,E1 25.1255,E2 411.8715} C_DIS
LIN {X 37.0505,Y 26.8869,Z 67,A 28.4053,B 24.8445,C -2.877,E1 25.1306,E2 414.9512} C_DIS
LIN {X 38.3748,Y 24.961,Z 67,A 25.5348,B 24.8452,C -2.8707,E1 25.1351,E2 417.8224} C_DIS
LIN {X 39.5207,Y 23.1034,Z 67,A 22.7971,B 24.8459,C -2.8635,E1 25.139,E2 420.5631} C_DIS
LIN {X 40.6422,Y 21.0686,Z 67,A 19.9558,B 24.8466,C -2.857,E1 25.1428,E2 423.4051} C_DIS
LIN {X 41.5991,Y 19.1095,Z 67,A 17.2724,B 24.8474,C -2.8503,E1 25.146,E2 426.0898} C_DIS
LIN {X 42.4841,Y 17.0516,Z 67,A 14.4301,B 24.8483,C -2.8417,E1 25.149,E2 428.9368} C_DIS
LIN {X 43.2874,Y 14.8956,Z 67,A 11.5767,B 24.8491,C -2.8338,E1 25.1517,E2 431.7928} C_DIS
LIN {X 43.9546,Y 12.7927,Z 67,A 8.8059,B 24.85,C -2.8255,E1 25.154,E2 434.5675} C_DIS
LIN {X 44.5243,Y 10.6413,Z 67,A 6.0409,B 24.8509,C -2.8176,E1 25.1559,E2 437.3353} C_DIS
LIN {X 44.9885,Y 8.4661,Z 67,A 3.2631,B 24.8518,C -2.8092,E1 25.1574,E2 440.1167} C_DIS
LIN {X 45.3427,Y 6.298,Z 67,A 0.5292,B 24.8526,C -2.8011,E1 25.1585,E2 442.8538} C_DIS
LIN {X 45.6043,Y 3.9869,Z 67,A -2.348,B 24.8535,C -2.7926,E1 25.1593,E2 445.7339} C_DIS
LIN {X 45.7449,Y 1.7478,Z 67,A -5.1153,B 24.8543,C -2.7846,E1 25.1597,E2 448.5038} C_DIS
LIN {X 45.7748,Y -0.5844,Z 67,A -7.8366,B 24.8549,C -2.7791,E1 25.1597,E2 451.2219} C_DIS
LIN {X 45.6993,Y -2.6839,Z 67,A -10.6374,B 24.8561,C -2.7676,E1 25.1594,E2 454.0331} C_DIS
LIN {X 45.5032,Y -5.0124,Z 67,A -13.527,B 24.857,C -2.7591,E1 25.1586,E2 456.9259} C_DIS
LIN {X 45.1946,Y -7.2885,Z 67,A -16.354,B 24.8579,C -2.7509,E1 25.1574,E2 459.7556} C_DIS
LIN {X 44.7844,Y -9.4886,Z 67,A -19.1404,B 24.8587,C -2.7425,E1 25.1559,E2 462.5458} C_DIS
LIN {X 44.273,Y -11.6435,Z 67,A -21.9042,B 24.8596,C -2.734,E1 25.1541,E2 465.3135} C_DIS
LIN {X 43.6615,Y -13.7593,Z 67,A -24.6752,B 24.8605,C -2.7253,E1 25.1518,E2 468.0894} C_DIS
LIN {X 42.937,Y -15.8764,Z 67,A -27.4347,B 24.8613,C -2.7175,E1 25.1492,E2 470.8517} C_DIS
LIN {X 42.0772,Y -18.0329,Z 67,A -30.2786,B 24.8621,C -2.71,E1 25.1462,E2 473.6978} C_DIS
LIN {X 41.1649,Y -20.0276,Z 67,A -33.1037,B 24.8631,C -2.7004,E1 25.1428,E2 476.5302} C_DIS
LIN {X 40.0773,Y -22.1238,Z 67,A -35.9288,B 24.8637,C -2.6943,E1 25.1391,E2 479.3549} C_DIS
LIN {X 38.9655,Y -24.0283,Z 67,A -38.696,B 24.8645,C -2.6864,E1 25.1351,E2 482.1267} C_DIS
LIN {X 37.7752,Y -25.859,Z 67,A -41.5204,B 24.8654,C -2.6773,E1 25.1308,E2 484.9587} C_DIS
LIN {X 36.2768,Y -27.9213,Z 67,A -44.6338,B 24.8661,C -2.6702,E1 25.1256,E2 488.0739} C_DIS
LIN {X 34.8671,Y -29.6629,Z 67,A -47.4223,B 24.8668,C -2.6633,E1 25.1206,E2 490.8659} C_DIS
LIN {X 33.3741,Y -31.3333,Z 67,A -50.1918,B 24.8674,C -2.657,E1 25.1153,E2 493.6381} C_DIS
LIN {X 31.7812,Y -32.9478,Z 67,A -53.0155,B 24.8681,C -2.6506,E1 25.1097,E2 496.4652} C_DIS
LIN {X 30.1087,Y -34.4829,Z 67,A -55.8428,B 24.8687,C -2.6444,E1 25.1038,E2 499.2958} C_DIS
LIN {X 28.2859,Y -35.9934,Z 67,A -58.8634,B 24.8694,C -2.637,E1 25.0973,E2 502.3226} C_DIS
LIN {X 26.3281,Y -37.4499,Z 67,A -61.8176,B 24.8699,C -2.6325,E1 25.0906,E2 505.2769} C_DIS
LIN {X 24.4881,Y -38.6783,Z 67,A -64.5643,B 24.8704,C -2.6276,E1 25.0842,E2 508.0261} C_DIS
LIN {X 22.5891,Y -39.8171,Z 67,A -67.3408,B 24.8709,C -2.6226,E1 25.0775,E2 510.8061} C_DIS
LIN {X 20.5833,Y -40.8902,Z 67,A -70.1873,B 24.8713,C -2.6179,E1 25.0704,E2 513.6558} C_DIS
LIN {X 18.5997,Y -41.8295,Z 67,A -72.9331,B 24.8717,C -2.6138,E1 25.0634,E2 516.4046} C_DIS
LIN {X 16.4549,Y -42.7189,Z 67,A -75.8195,B 24.8721,C -2.6101,E1 25.0559,E2 519.2932} C_DIS
LIN {X 14.4039,Y -43.4533,Z 67,A -78.5659,B 24.8725,C -2.6064,E1 25.0487,E2 522.043} C_DIS
LIN {X 12.2045,Y -44.1217,Z 67,A -81.3883,B 24.8727,C -2.6041,E1 25.0411,E2 524.8659} C_DIS
LIN {X 10.0324,Y -44.6658,Z 67,A -84.188,B 24.8729,C -2.6015,E1 25.0335,E2 527.6678} C_DIS
LIN {X 7.7901,Y -45.1107,Z 67,A -87.1251,B 24.8733,C -2.598,E1 25.0254,E2 530.6099} C_DIS
LIN {X 5.5161,Y -45.4446,Z 67,A -89.9049,B 24.8733,C -2.5977,E1 25.0177,E2 533.3881} C_DIS
LIN {X 3.3464,Y -45.656,Z 67,A -92.6178,B 24.8734,C -2.5966,E1 25.0102,E2 536.1022} C_DIS
LIN {X 1.1515,Y -45.764,Z 67,A -95.4014,B 24.8736,C -2.5951,E1 25.0024,E2 538.8885} C_DIS
LIN {X 1.1515,Y -45.764,Z 67,A -95.4014,B 24.8736,C -2.5951,E1 25.0024,E2 538.8885} C_DIS
Enddeposition()
LIN {X 0.2417,Y -47.8891,Z 71.5315,A -95.4317,B 24.8723,C -2.6079,E1 25.0024,E2 538.8885} C_DIS
LIN {X 0.3246,Y -54.2279,Z 85.1262,A -95.401,B 24.8736,C -2.595,E1 25.0024,E2 538.8885} C_DIS
LIN {X 0.3246,Y -54.2279,Z 106.1262,A -95.7537,B 24.8587,C -2.7433,E1 25.0024,E2 538.8885} C_DIS
LIN {X 0.4528,Y -68.2127,Z 106.1262,A -95.2481,B 24.8816,C -2.5114,E1 25.0023,E2 538.9342} C_DIS
LIN {X 0.4528,Y -68.2127,Z 86.1262,A -94.9125,B 24.8946,C -2.3702,E1 25.0023,E2 538.9342} C_DIS
LIN {X 0.375,Y -61.8739,Z 72.5315,A -94.9409,B 24.8935,C -2.3821,E1 25.0023,E2 538.9342} C_DIS
LIN {X 0.3491,Y -59.761,Z 68,A -94.9519,B 24.8931,C -2.3867,E1 25.0023,E2 538.9342} C_DIS
Startdeposition()
$VEL.CP = VEL_PRINT
LIN {X 2.9325,Y -59.6933,Z 68,A -92.1575,B 24.8924,C -2.3943,E1 25.0101,E2 536.1226} C_DIS
LIN {X 5.858,Y -59.4775,Z 68,A -89.3481,B 24.8923,C -2.3957,E1 25.0179,E2 533.3115} C_DIS
LIN {X 8.7694,Y -59.1184,Z 68,A -86.5399,B 24.8921,C -2.3974,E1 25.0257,E2 530.5015} C_DIS
LIN {X 11.6596,Y -58.6169,Z 68,A -83.7325,B 24.8919,C -2.3996,E1 25.0334,E2 527.6921} C_DIS
LIN {X 14.5218,Y -57.9742,Z 68,A -80.926,B 24.8917,C -2.4021,E1 25.0411,E2 524.8836} C_DIS
LIN {X 17.3489,Y -57.1918,Z 68,A -78.1205,B 24.8914,C -2.4051,E1 25.0486,E2 522.0759} C_DIS
LIN {X 20.1343,Y -56.2716,Z 68,A -75.316,B 24.8911,C -2.4084,E1 25.056,E2 519.269} C_DIS
LIN {X 22.8712,Y -55.2159,Z 68,A -72.5122,B 24.8908,C -2.4121,E1 25.0633,E2 516.4628} C_DIS
LIN {X 25.5529,Y -54.0272,Z 68,A -69.7093,B 24.8904,C -2.4162,E1 25.0704,E2 513.6574} C_DIS
LIN {X 28.1732,Y -52.7083,Z 68,A -66.9073,B 24.89,C -2.4206,E1 25.0773,E2 510.8526} C_DIS
LIN {X 30.7255,Y -51.2624,Z 68,A -64.1063,B 24.8896,C -2.4254,E1 25.0841,E2 508.0489} C_DIS
LIN {X 33.2038,Y -49.693,Z 68,A -61.3059,B 24.8891,C -2.4305,E1 25.0907,E2 505.2456} C_DIS
LIN {X 35.6021,Y -48.0039,Z 68,A -58.5063,B 24.8886,C -2.4359,E1 25.097,E2 502.443} C_DIS
LIN {X 37.9147,Y -46.1992,Z 68,A -55.7074,B 24.8881,C -2.4416,E1 25.1031,E2 499.641} C_DIS
LIN {X 40.1359,Y -44.2831,Z 68,A -52.9092,B 24.8876,C -2.4477,E1 25.109,E2 496.8396} C_DIS
LIN {X 42.2604,Y -42.2604,Z 68,A -50.1117,B 24.887,C -2.454,E1 25.1146,E2 494.0389} C_DIS
LIN {X 44.2831,Y -40.1359,Z 68,A -47.3149,B 24.8864,C -2.4606,E1 25.1199,E2 491.2388} C_DIS
LIN {X 46.1992,Y -37.9147,Z 68,A -44.5186,B 24.8857,C -2.4674,E1 25.1249,E2 488.4392} C_DIS
LIN {X 48.0039,Y -35.6021,Z 68,A -41.7229,B 24.8851,C -2.4744,E1 25.1296,E2 485.6401} C_DIS
LIN {X 49.693,Y -33.2038,Z 68,A -38.9276,B 24.8844,C -2.4817,E1 25.1341,E2 482.8414} C_DIS
LIN {X 51.2624,Y -30.7255,Z 68,A -36.1328,B 24.8837,C -2.4892,E1 25.1382,E2 480.0431} C_DIS
LIN {X 52.7083,Y -28.1732,Z 68,A -33.3384,B 24.883,C -2.4968,E1 25.1419,E2 477.2453} C_DIS
LIN {X 54.0312,Y -25.5443,Z 68,A -30.5419,B 24.8823,C -2.5045,E1 25.1454,E2 474.4456} C_DIS
LIN {X 55.2159,Y -22.8712,Z 68,A -27.751,B 24.8815,C -2.5126,E1 25.1484,E2 471.6508} C_DIS
LIN {X 56.2716,Y -20.1343,Z 68,A -24.9577,B 24.8807,C -2.5207,E1 25.1511,E2 468.854} C_DIS
LIN {X 57.1918,Y -17.3489,Z 68,A -22.1646,B 24.88,C -2.5288,E1 25.1535,E2 466.0575} C_DIS
LIN {X 57.9742,Y -14.5218,Z 68,A -19.3717,B 24.8792,C -2.5371,E1 25.1555,E2 463.2611} C_DIS
LIN {X 58.6169,Y -11.6596,Z 68,A -16.5792,B 24.8784,C -2.5455,E1 25.1571,E2 460.4651} C_DIS
LIN {X 59.1184,Y -8.7694,Z 68,A -13.7864,B 24.8776,C -2.5538,E1 25.1583,E2 457.669} C_DIS
LIN {X 59.4775,Y -5.858,Z 68,A -10.994,B 24.8768,C -2.5622,E1 25.1592,E2 454.8732} C_DIS
LIN {X 59.6933,Y -2.9325,Z 68,A -8.2015,B 24.8759,C -2.5707,E1 25.1597,E2 452.0774} C_DIS
LIN {X 59.7608,Y -0.7334,Z 68,A -6.3075,B 24.8758,C -2.5721,E1 25.1597,E2 450.1912} C_DIS
LIN {X 59.7337,Y 1.9101,Z 68,A -3.6601,B 24.8748,C -2.5828,E1 25.1597,E2 447.5342} C_DIS
LIN {X 59.5802,Y 4.6855,Z 68,A -1.1251,B 24.8742,C -2.5881,E1 25.1592,E2 445.0019} C_DIS
LIN {X 59.3158,Y 7.3159,Z 68,A 1.5727,B 24.8731,C -2.5999,E1 25.1583,E2 442.2922} C_DIS
LIN {X 58.8854,Y 10.2176,Z 68,A 4.3658,B 24.8723,C -2.6081,E1 25.1571,E2 439.4961} C_DIS
LIN {X 58.3131,Y 13.0946,Z 68,A 7.159,B 24.8715,C -2.6162,E1 25.1555,E2 436.7} C_DIS
LIN {X 57.6003,Y 15.9402,Z 68,A 9.9525,B 24.8707,C -2.6242,E1 25.1535,E2 433.9037} C_DIS
LIN {X 56.7488,Y 18.7473,Z 68,A 12.7464,B 24.8699,C -2.632,E1 25.1511,E2 431.1071} C_DIS
LIN {X 55.7606,Y 21.5092,Z 68,A 15.5407,B 24.8692,C -2.6397,E1 25.1484,E2 428.3102} C_DIS
LIN {X 54.638,Y 24.2194,Z 68,A 18.3353,B 24.8684,C -2.6472,E1 25.1453,E2 425.5132} C_DIS
LIN {X 53.3838,Y 26.8711,Z 68,A 21.1304,B 24.8677,C -2.6545,E1 25.1419,E2 422.7158} C_DIS
LIN {X 52.001,Y 29.4582,Z 68,A 23.9261,B 24.867,C -2.6616,E1 25.1381,E2 419.918} C_DIS
LIN {X 50.4929,Y 31.9743,Z 68,A 26.7223,B 24.8663,C -2.6685,E1 25.134,E2 417.1197} C_DIS
LIN {X 48.8632,Y 34.4133,Z 68,A 29.519,B 24.8656,C -2.6751,E1 25.1296,E2 414.3211} C_DIS
LIN {X 47.1157,Y 36.7695,Z 68,A 32.3164,B 24.865,C -2.6814,E1 25.1248,E2 411.5219} C_DIS
LIN {X 45.2548,Y 39.0371,Z 68,A 35.1144,B 24.8644,C -2.6875,E1 25.1198,E2 408.7223} C_DIS
LIN {X 43.2848,Y 41.2106,Z 68,A 37.9132,B 24.8638,C -2.6933,E1 25.1145,E2 405.9221} C_DIS
LIN {X 41.2106,Y 43.2848,Z 68,A 40.7125,B 24.8632,C -2.6988,E1 25.1089,E2 403.1214} C_DIS
LIN {X 39.0371,Y 45.2548,Z 68,A 43.5128,B 24.8627,C -2.704,E1 25.103,E2 400.32} C_DIS
LIN {X 36.7695,Y 47.1157,Z 68,A 46.3137,B 24.8622,C -2.7088,E1 25.0969,E2 397.5181} C_DIS
LIN {X 34.4133,Y 48.8632,Z 68,A 49.1154,B 24.8617,C -2.7133,E1 25.0906,E2 394.7156} C_DIS
LIN {X 31.9743,Y 50.4929,Z 68,A 51.9182,B 24.8613,C -2.7175,E1 25.084,E2 391.9122} C_DIS
LIN {X 29.4582,Y 52.001,Z 68,A 54.7216,B 24.8609,C -2.7213,E1 25.0772,E2 389.1083} C_DIS
LIN {X 26.8711,Y 53.3838,Z 68,A 57.526,B 24.8606,C -2.7247,E1 25.0703,E2 386.3036} C_DIS
LIN {X 24.2194,Y 54.638,Z 68,A 60.3593,B 24.8602,C -2.7283,E1 25.0631,E2 383.4687} C_DIS
LIN {X 21.5092,Y 55.7606,Z 68,A 63.1375,B 24.86,C -2.7303,E1 25.0559,E2 380.692} C_DIS
LIN {X 18.7473,Y 56.7488,Z 68,A 65.9447,B 24.8598,C -2.7326,E1 25.0485,E2 377.885} C_DIS
LIN {X 15.9402,Y 57.6003,Z 68,A 68.7527,B 24.8596,C -2.7344,E1 25.041,E2 375.0774} C_DIS
LIN {X 13.0946,Y 58.3131,Z 68,A 71.5619,B 24.8594,C -2.7359,E1 25.0333,E2 372.2688} C_DIS
LIN {X 10.2176,Y 58.8854,Z 68,A 74.3719,B 24.8594,C -2.7369,E1 25.0256,E2 369.4595} C_DIS
LIN {X 7.3159,Y 59.3158,Z 68,A 77.1828,B 24.8592,C -2.7375,E1 25.0178,E2 366.6494} C_DIS
LIN {X 4.3966,Y 59.6033,Z 68,A 79.995,B 24.8592,C -2.7377,E1 25.01,E2 363.8384} C_DIS
LIN {X 1.4667,Y 59.7473,Z 68,A 82.8079,B 24.8592,C -2.7375,E1 25.0022,E2 361.0266} C_DIS
LIN {X -1.4667,Y 59.7473,Z 68,A 85.6322,B 24.8592,C -2.7371,E1 24.9943,E2 358.2032} C_DIS
LIN {X -4.3966,Y 59.6033,Z 68,A 88.4369,B 24.8594,C -2.7359,E1 24.9865,E2 355.4006} C_DIS
LIN {X -7.3159,Y 59.3158,Z 68,A 91.2527,B 24.8596,C -2.7344,E1 24.9787,E2 352.5865} C_DIS
LIN {X -10.2176,Y 58.8854,Z 68,A 94.0698,B 24.8598,C -2.7326,E1 24.9709,E2 349.7712} C_DIS
LIN {X -13.0946,Y 58.3131,Z 68,A 96.8875,B 24.86,C -2.7303,E1 24.9632,E2 346.9555} C_DIS
LIN {X -15.9402,Y 57.6003,Z 68,A 99.7064,B 24.8603,C -2.7277,E1 24.9556,E2 344.1387} C_DIS
LIN {X -18.7473,Y 56.7488,Z 68,A 102.5262,B 24.8606,C -2.7246,E1 24.9481,E2 341.3212} C_DIS
LIN {X -21.5092,Y 55.7606,Z 68,A 105.3469,B 24.8609,C -2.7212,E1 24.9407,E2 338.5029} C_DIS
LIN {X -24.2194,Y 54.638,Z 68,A 108.1684,B 24.8613,C -2.7174,E1 24.9335,E2 335.6839} C_DIS
LIN {X -26.8711,Y 53.3838,Z 68,A 110.9908,B 24.8618,C -2.7132,E1 24.9264,E2 332.8641} C_DIS
LIN {X -29.4582,Y 52.001,Z 68,A 113.8142,B 24.8622,C -2.7086,E1 24.9195,E2 330.0435} C_DIS
LIN {X -31.9743,Y 50.4929,Z 68,A 116.6383,B 24.8627,C -2.7037,E1 24.9128,E2 327.2221} C_DIS
LIN {X -34.4133,Y 48.8632,Z 68,A 119.4633,B 24.8632,C -2.6985,E1 24.9063,E2 324.4002} C_DIS
LIN {X -36.7695,Y 47.1157,Z 68,A 122.289,B 24.8638,C -2.693,E1 24.9001,E2 321.5774} C_DIS
LIN {X -39.0371,Y 45.2548,Z 68,A 125.1154,B 24.8644,C -2.6871,E1 24.894,E2 318.7541} C_DIS
LIN {X -41.2106,Y 43.2848,Z 68,A 127.9426,B 24.865,C -2.6809,E1 24.8882,E2 315.9302} C_DIS
LIN {X -43.2848,Y 41.2106,Z 68,A 130.7704,B 24.8657,C -2.6745,E1 24.8827,E2 313.1056} C_DIS
LIN {X -45.2548,Y 39.0371,Z 68,A 133.5989,B 24.8664,C -2.6678,E1 24.8775,E2 310.2805} C_DIS
LIN {X -47.1157,Y 36.7695,Z 68,A 136.4279,B 24.8671,C -2.6608,E1 24.8726,E2 307.4548} C_DIS
LIN {X -48.8632,Y 34.4133,Z 68,A 139.2576,B 24.8678,C -2.6536,E1 24.868,E2 304.6286} C_DIS
LIN {X -50.4929,Y 31.9743,Z 68,A 142.0877,B 24.8685,C -2.6462,E1 24.8637,E2 301.8019} C_DIS
LIN {X -52.001,Y 29.4582,Z 68,A 144.9182,B 24.8693,C -2.6386,E1 24.8597,E2 298.9749} C_DIS
LIN {X -53.3838,Y 26.8711,Z 68,A 147.7493,B 24.87,C -2.6308,E1 24.8561,E2 296.1473} C_DIS
LIN {X -54.638,Y 24.2194,Z 68,A 150.5807,B 24.8708,C -2.6229,E1 24.8528,E2 293.3195} C_DIS
LIN {X -55.7606,Y 21.5092,Z 68,A 153.4124,B 24.8716,C -2.6148,E1 24.8498,E2 290.4912} C_DIS
LIN {X -56.7488,Y 18.7473,Z 68,A 156.2443,B 24.8724,C -2.6066,E1 24.8473,E2 287.6628} C_DIS
LIN {X -57.6003,Y 15.9402,Z 68,A 159.0767,B 24.8733,C -2.5982,E1 24.8451,E2 284.8339} C_DIS
LIN {X -58.3131,Y 13.0946,Z 68,A 161.909,B 24.8741,C -2.5899,E1 24.8433,E2 282.0051} C_DIS
LIN {X -58.8854,Y 10.2176,Z 68,A 164.7417,B 24.8749,C -2.5814,E1 24.8418,E2 279.1758} C_DIS
LIN {X -59.3158,Y 7.3159,Z 68,A 167.5743,B 24.8757,C -2.5729,E1 24.8408,E2 276.3466} C_DIS
LIN {X -59.6033,Y 4.3966,Z 68,A 170.4072,B 24.8765,C -2.5644,E1 24.8401,E2 273.5171} C_DIS
LIN {X -59.7473,Y 1.4667,Z 68,A 173.1568,B 24.8775,C -2.5544,E1 24.8398,E2 270.7748} C_DIS
LIN {X -59.7473,Y -1.4667,Z 68,A 176.0726,B 24.8782,C -2.5474,E1 24.8398,E2 267.8583} C_DIS
LIN {X -59.6033,Y -4.3966,Z 68,A 178.9052,B 24.879,C -2.5389,E1 24.8404,E2 265.0288} C_DIS
LIN {X -59.3158,Y -7.3159,Z 68,A -178.2625,B 24.8798,C -2.5306,E1 24.8413,E2 262.1996} C_DIS
LIN {X -58.8854,Y -10.2176,Z 68,A -175.4301,B 24.8806,C -2.5223,E1 24.8425,E2 259.3702} C_DIS
LIN {X -58.3131,Y -13.0946,Z 68,A -172.5983,B 24.8814,C -2.5141,E1 24.8441,E2 256.5412} C_DIS
LIN {X -57.6003,Y -15.9402,Z 68,A -169.7666,B 24.8821,C -2.506,E1 24.8462,E2 253.7123} C_DIS
LIN {X -56.7488,Y -18.7473,Z 68,A -166.9352,B 24.8829,C -2.4981,E1 24.8486,E2 250.8836} C_DIS
LIN {X -55.7606,Y -21.5092,Z 68,A -164.1042,B 24.8836,C -2.4903,E1 24.8513,E2 248.0552} C_DIS
LIN {X -54.638,Y -24.2194,Z 68,A -161.2738,B 24.8843,C -2.4827,E1 24.8544,E2 245.2272} C_DIS
LIN {X -53.3838,Y -26.8711,Z 68,A -158.4438,B 24.885,C -2.4754,E1 24.8579,E2 242.3996} C_DIS
LIN {X -52.001,Y -29.4582,Z 68,A -155.6143,B 24.8857,C -2.4682,E1 24.8617,E2 239.5722} C_DIS
LIN {X -50.4929,Y -31.9743,Z 68,A -152.7853,B 24.8863,C -2.4613,E1 24.8658,E2 236.7453} C_DIS
Enddeposition()
END
